   1:  PR[GP1:91,2] = PR[GP1:90,2] + 17.555;
   1:L PR[91] R[100]mm/sec CNT100;
   1:  PR[GP1:91,1] = PR[GP1:90,1] + 68.988;
   1:  PR[GP1:91,2] = PR[GP1:90,2] + 18.519;
   1:L PR[91] R[100]mm/sec CNT100;
   1:  PR[GP1:91,1] = PR[GP1:90,1] + 65.480;
   1:  PR[GP1:91,2] = PR[GP1:90,2] + 23.094;
   1:L PR[91] R[100]mm/sec CNT100;
   1:  PR[GP1:91,1] = PR[GP1:90,1] + 60.307;
   1:  PR[GP1:91,2] = PR[GP1:90,2] + 27.735;
   1:L PR[91] R[100]mm/sec CNT100;
   1:  PR[GP1:91,1] = PR[GP1:90,1] + 55.410;
   1:  PR[GP1:91,2] = PR[GP1:90,2] + 30.688;
   1:L PR[91] R[100]mm/sec CNT100;
   1:  PR[GP1:91,1] = PR[GP1:90,1] + 49.981;
   1:  PR[GP1:91,2] = PR[GP1:90,2] + 32.704;
   1:L PR[91] R[100]mm/sec CNT100;
   1:  PR[GP1:91,1] = PR[GP1:90,1] + 48.884;
   1:  PR[GP1:91,2] = PR[GP1:90,2] + 33.180;
   1:L PR[91] R[100]mm/sec CNT100;
   1:  PR[GP1:91,1] = PR[GP1:90,1] + 43.284;
   1:  PR[GP1:91,2] = PR[GP1:90,2] + 34.134;
   1:L PR[91] R[100]mm/sec CNT100;
   1:  PR[GP1:91,1] = PR[GP1:90,1] + 41.949;
   1:  PR[GP1:91,2] = PR[GP1:90,2] + 34.234;
   1:L PR[91] R[100]mm/sec CNT100;
   1:  PR[GP1:91,1] = PR[GP1:90,1] + 36.318;
   1:  PR[GP1:91,2] = PR[GP1:90,2] + 34.132;
   1:L PR[91] R[100]mm/sec CNT100;
   1:  PR[GP1:91,1] = PR[GP1:90,1] + 30.791;
   1:  PR[GP1:91,2] = PR[GP1:90,2] + 32.982;
   1:L PR[91] R[100]mm/sec CNT100;
   1:  PR[GP1:91,1] = PR[GP1:90,1] + 29.393;
   1:  PR[GP1:91,2] = PR[GP1:90,2] + 32.616;
   1:L PR[91] R[100]mm/sec CNT100;
   1:  PR[GP1:91,1] = PR[GP1:90,1] + 24.268;
   1:  PR[GP1:91,2] = PR[GP1:90,2] + 30.497;
   1:L PR[91] R[100]mm/sec CNT100;
   1:  PR[GP1:91,1] = PR[GP1:90,1] + 18.293;
   1:  PR[GP1:91,2] = PR[GP1:90,2] + 26.578;
   1:L PR[91] R[100]mm/sec CNT100;
   1:  PR[GP1:91,1] = PR[GP1:90,1] + 14.361;
   1:  PR[GP1:91,2] = PR[GP1:90,2] + 22.795;
   1:L PR[91] R[100]mm/sec CNT100;
   1:  PR[GP1:91,1] = PR[GP1:90,1] + 11.161;
   1:  PR[GP1:91,2] = PR[GP1:90,2] + 18.294;
   1:L PR[91] R[100]mm/sec CNT100;
   1:  PR[GP1:91,1] = PR[GP1:90,1] + 10.144;
   1:  PR[GP1:91,2] = PR[GP1:90,2] + 16.966;
   1:L PR[91] R[100]mm/sec CNT100;
   1:  PR[GP1:91,1] = PR[GP1:90,1] + 7.887;
   1:  PR[GP1:91,2] = PR[GP1:90,2] + 12.055;
   1:L PR[91] R[100]mm/sec CNT100;
   1:  PR[GP1:91,1] = PR[GP1:90,1] + 7.315;
   1:  PR[GP1:91,2] = PR[GP1:90,2] + 10.330;
   1:L PR[91] R[100]mm/sec CNT100;
   1:  PR[GP1:91,1] = PR[GP1:90,1] + 6.110;
   1:  PR[GP1:91,2] = PR[GP1:90,2] + 5.493;
   1:L PR[91] R[100]mm/sec CNT100;
   1:  PR[GP1:91,1] = PR[GP1:90,1] + 6.265;
   1:  PR[GP1:91,2] = PR[GP1:90,2] + 5.404;
   1:L PR[91] R[100]mm/sec CNT100;
   1:  PR[GP1:91,1] = PR[GP1:90,1] + 4.352;
   1:  PR[GP1:91,2] = PR[GP1:90,2] + 1.921;
   1:L PR[91] R[100]mm/sec CNT100;
   1:  PR[GP1:91,1] = PR[GP1:90,1] + 4.139;
   1:  PR[GP1:91,2] = PR[GP1:90,2] + 1.690;
   1:L PR[91] R[100]mm/sec CNT100;
   1:  PR[GP1:91,1] = PR[GP1:90,1] + 3.838;
   1:  PR[GP1:91,2] = PR[GP1:90,2] + 1.482;
   1:L PR[91] R[100]mm/sec CNT100;
   1:  PR[GP1:91,1] = PR[GP1:90,1] + 1.067;
   1:  PR[GP1:91,2] = PR[GP1:90,2] + 0.455;
   1:L PR[91] R[100]mm/sec CNT100;
   1:  PR[GP1:91,1] = PR[GP1:90,1] + 0.591;
   1:  PR[GP1:91,2] = PR[GP1:90,2] + 0.328;
   1:L PR[91] R[100]mm/sec CNT100;
   1:  PR[GP1:91,1] = PR[GP1:90,1] + -0.408;
   1:L PR[91] R[100]mm/sec CNT100;
   1:  ! -- Layer/Ebene 16 -- !;
   1:  PR[91] = PR[90];
   1:  PR[GP1:91,1] = PR[GP1:90,1] + -1.944;
   1:  PR[GP1:91,2] = PR[GP1:90,2] + 0.906;
   1:  PR[GP1:91,3] = PR[GP1:90,3] + 10.065;
   1:L PR[91] R[100]mm/sec CNT100;
   1:  PR[GP1:91,1] = PR[GP1:90,1] + -2.665;
   1:  PR[GP1:91,2] = PR[GP1:90,2] + 1.194;
   1:L PR[91] R[100]mm/sec CNT100;
   1:  PR[GP1:91,1] = PR[GP1:90,1] + -2.731;
   1:  PR[GP1:91,2] = PR[GP1:90,2] + 1.197;
   1:L PR[91] R[100]mm/sec CNT100;
   1:  PR[GP1:91,1] = PR[GP1:90,1] + -3.897;
   1:  PR[GP1:91,2] = PR[GP1:90,2] + 1.658;
   1:L PR[91] R[100]mm/sec CNT100;
   1:  PR[GP1:91,1] = PR[GP1:90,1] + -5.226;
   1:  PR[GP1:91,2] = PR[GP1:90,2] + 4.059;
   1:L PR[91] R[100]mm/sec CNT100;
   1:  PR[GP1:91,1] = PR[GP1:90,1] + -6.062;
   1:  PR[GP1:91,2] = PR[GP1:90,2] + 5.392;
   1:L PR[91] R[100]mm/sec CNT100;
   1:  PR[GP1:91,1] = PR[GP1:90,1] + -5.854;
   1:  PR[GP1:91,2] = PR[GP1:90,2] + 5.510;
   1:L PR[91] R[100]mm/sec CNT100;
   1:  PR[GP1:91,1] = PR[GP1:90,1] + -6.919;
   1:  PR[GP1:91,2] = PR[GP1:90,2] + 9.788;
   1:L PR[91] R[100]mm/sec CNT100;
   1:  PR[GP1:91,1] = PR[GP1:90,1] + -7.804;
   1:  PR[GP1:91,2] = PR[GP1:90,2] + 12.458;
   1:L PR[91] R[100]mm/sec CNT100;
   1:  PR[GP1:91,1] = PR[GP1:90,1] + -9.839;
   1:  PR[GP1:91,2] = PR[GP1:90,2] + 16.883;
   1:L PR[91] R[100]mm/sec CNT100;
   1:  PR[GP1:91,1] = PR[GP1:90,1] + -12.674;
   1:  PR[GP1:91,2] = PR[GP1:90,2] + 20.871;
   1:L PR[91] R[100]mm/sec CNT100;
   1:  PR[GP1:91,1] = PR[GP1:90,1] + -14.304;
   1:  PR[GP1:91,2] = PR[GP1:90,2] + 23.006;
   1:L PR[91] R[100]mm/sec CNT100;
   1:  PR[GP1:91,1] = PR[GP1:90,1] + -17.875;
   1:  PR[GP1:91,2] = PR[GP1:90,2] + 26.441;
   1:L PR[91] R[100]mm/sec CNT100;
   1:  PR[GP1:91,1] = PR[GP1:90,1] + -22.062;
   1:  PR[GP1:91,2] = PR[GP1:90,2] + 29.178;
   1:L PR[91] R[100]mm/sec CNT100;
   1:  PR[GP1:91,1] = PR[GP1:90,1] + -24.170;
   1:  PR[GP1:91,2] = PR[GP1:90,2] + 30.576;
   1:L PR[91] R[100]mm/sec CNT100;
   1:  PR[GP1:91,1] = PR[GP1:90,1] + -28.843;
   1:  PR[GP1:91,2] = PR[GP1:90,2] + 32.508;
   1:L PR[91] R[100]mm/sec CNT100;
   1:  PR[GP1:91,1] = PR[GP1:90,1] + -33.865;
   1:  PR[GP1:91,2] = PR[GP1:90,2] + 33.553;
   1:L PR[91] R[100]mm/sec CNT100;
   1:  PR[GP1:91,1] = PR[GP1:90,1] + -36.143;
   1:  PR[GP1:91,2] = PR[GP1:90,2] + 34.143;
   1:L PR[91] R[100]mm/sec CNT100;
   1:  PR[GP1:91,1] = PR[GP1:90,1] + -41.327;
   1:  PR[GP1:91,2] = PR[GP1:90,2] + 34.237;
   1:L PR[91] R[100]mm/sec CNT100;
   1:  PR[GP1:91,1] = PR[GP1:90,1] + -43.399;
   1:  PR[GP1:91,2] = PR[GP1:90,2] + 34.081;
   1:L PR[91] R[100]mm/sec CNT100;
   1:  PR[GP1:91,1] = PR[GP1:90,1] + -48.621;
   1:  PR[GP1:91,2] = PR[GP1:90,2] + 33.191;
   1:L PR[91] R[100]mm/sec CNT100;
   1:  PR[GP1:91,1] = PR[GP1:90,1] + -53.599;
   1:  PR[GP1:91,2] = PR[GP1:90,2] + 31.342;
   1:L PR[91] R[100]mm/sec CNT100;
   1:  PR[GP1:91,1] = PR[GP1:90,1] + -55.379;
   1:  PR[GP1:91,2] = PR[GP1:90,2] + 30.575;
   1:L PR[91] R[100]mm/sec CNT100;
   1:  PR[GP1:91,1] = PR[GP1:90,1] + -59.971;
   1:  PR[GP1:91,2] = PR[GP1:90,2] + 27.806;
   1:L PR[91] R[100]mm/sec CNT100;
   1:  PR[GP1:91,1] = PR[GP1:90,1] + -63.997;
   1:  PR[GP1:91,2] = PR[GP1:90,2] + 24.207;
   1:L PR[91] R[100]mm/sec CNT100;
   1:  PR[GP1:91,1] = PR[GP1:90,1] + -65.346;
   1:  PR[GP1:91,2] = PR[GP1:90,2] + 22.977;
   1:L PR[91] R[100]mm/sec CNT100;
   1:  PR[GP1:91,1] = PR[GP1:90,1] + -68.635;
   1:  PR[GP1:91,2] = PR[GP1:90,2] + 18.689;
   1:L PR[91] R[100]mm/sec CNT100;
   1:  PR[GP1:91,1] = PR[GP1:90,1] + -71.099;
   1:  PR[GP1:91,2] = PR[GP1:90,2] + 13.808;
   1:L PR[91] R[100]mm/sec CNT100;
   1:  PR[GP1:91,1] = PR[GP1:90,1] + -71.933;
   1:  PR[GP1:91,2] = PR[GP1:90,2] + 12.276;
   1:L PR[91] R[100]mm/sec CNT100;
   1:  PR[GP1:91,1] = PR[GP1:90,1] + -73.434;
   1:  PR[GP1:91,2] = PR[GP1:90,2] + 7.063;
   1:L PR[91] R[100]mm/sec CNT100;
   1:  PR[GP1:91,1] = PR[GP1:90,1] + -73.949;
   1:  PR[GP1:91,2] = PR[GP1:90,2] + 1.575;
   1:L PR[91] R[100]mm/sec CNT100;
   1:  PR[GP1:91,1] = PR[GP1:90,1] + -74.227;
   1:  PR[GP1:91,2] = PR[GP1:90,2] + -0.094;
   1:L PR[91] R[100]mm/sec CNT100;
   1:  PR[GP1:91,1] = PR[GP1:90,1] + -73.715;
   1:  PR[GP1:91,2] = PR[GP1:90,2] + -5.552;
   1:L PR[91] R[100]mm/sec CNT100;
   1:  PR[GP1:91,1] = PR[GP1:90,1] + -73.440;
   1:  PR[GP1:91,2] = PR[GP1:90,2] + -7.186;
   1:L PR[91] R[100]mm/sec CNT100;
   1:  PR[GP1:91,1] = PR[GP1:90,1] + -71.930;
   1:  PR[GP1:91,2] = PR[GP1:90,2] + -12.429;
   1:L PR[91] R[100]mm/sec CNT100;
   1:  PR[GP1:91,1] = PR[GP1:90,1] + -69.461;
   1:  PR[GP1:91,2] = PR[GP1:90,2] + -17.322;
   1:L PR[91] R[100]mm/sec CNT100;
   1:  PR[GP1:91,1] = PR[GP1:90,1] + -68.641;
   1:  PR[GP1:91,2] = PR[GP1:90,2] + -18.825;
   1:L PR[91] R[100]mm/sec CNT100;
   1:  PR[GP1:91,1] = PR[GP1:90,1] + -65.348;
   1:  PR[GP1:91,2] = PR[GP1:90,2] + -23.119;
   1:L PR[91] R[100]mm/sec CNT100;
   1:  PR[GP1:91,1] = PR[GP1:90,1] + -61.277;
   1:  PR[GP1:91,2] = PR[GP1:90,2] + -26.759;
   1:L PR[91] R[100]mm/sec CNT100;
   1:  PR[GP1:91,1] = PR[GP1:90,1] + -59.968;
   1:  PR[GP1:91,2] = PR[GP1:90,2] + -27.952;
   1:L PR[91] R[100]mm/sec CNT100;
   1:  PR[GP1:91,1] = PR[GP1:90,1] + -55.392;
   1:  PR[GP1:91,2] = PR[GP1:90,2] + -30.711;
   1:L PR[91] R[100]mm/sec CNT100;
   1:  PR[GP1:91,1] = PR[GP1:90,1] + -50.312;
   1:  PR[GP1:91,2] = PR[GP1:90,2] + -32.598;
   1:L PR[91] R[100]mm/sec CNT100;
   1:  PR[GP1:91,1] = PR[GP1:90,1] + -48.605;
   1:  PR[GP1:91,2] = PR[GP1:90,2] + -33.338;
   1:L PR[91] R[100]mm/sec CNT100;
   1:  PR[GP1:91,1] = PR[GP1:90,1] + -43.399;
   1:  PR[GP1:91,2] = PR[GP1:90,2] + -34.225;
   1:L PR[91] R[100]mm/sec CNT100;
   1:  PR[GP1:91,1] = PR[GP1:90,1] + -41.327;
   1:  PR[GP1:91,2] = PR[GP1:90,2] + -34.381;
   1:L PR[91] R[100]mm/sec CNT100;
   1:  PR[GP1:91,1] = PR[GP1:90,1] + -36.128;
   1:  PR[GP1:91,2] = PR[GP1:90,2] + -34.287;
   1:L PR[91] R[100]mm/sec CNT100;
   1:  PR[GP1:91,1] = PR[GP1:90,1] + -31.025;
   1:  PR[GP1:91,2] = PR[GP1:90,2] + -33.225;
   1:L PR[91] R[100]mm/sec CNT100;
   1:  PR[GP1:91,1] = PR[GP1:90,1] + -28.857;
   1:  PR[GP1:91,2] = PR[GP1:90,2] + -32.658;
   1:L PR[91] R[100]mm/sec CNT100;
   1:  PR[GP1:91,1] = PR[GP1:90,1] + -24.168;
   1:  PR[GP1:91,2] = PR[GP1:90,2] + -30.719;
   1:L PR[91] R[100]mm/sec CNT100;
   1:  PR[GP1:91,1] = PR[GP1:90,1] + -19.889;
   1:  PR[GP1:91,2] = PR[GP1:90,2] + -27.922;
   1:L PR[91] R[100]mm/sec CNT100;
   1:  PR[GP1:91,1] = PR[GP1:90,1] + -17.877;
   1:  PR[GP1:91,2] = PR[GP1:90,2] + -26.586;
   1:L PR[91] R[100]mm/sec CNT100;
   1:  PR[GP1:91,1] = PR[GP1:90,1] + -14.312;
   1:  PR[GP1:91,2] = PR[GP1:90,2] + -23.157;
   1:L PR[91] R[100]mm/sec CNT100;
   1:  PR[GP1:91,1] = PR[GP1:90,1] + -11.409;
   1:  PR[GP1:91,2] = PR[GP1:90,2] + -19.073;
   1:L PR[91] R[100]mm/sec CNT100;
   1:  PR[GP1:91,1] = PR[GP1:90,1] + -9.834;
   1:  PR[GP1:91,2] = PR[GP1:90,2] + -17.017;
   1:L PR[91] R[100]mm/sec CNT100;
   1:  PR[GP1:91,1] = PR[GP1:90,1] + -7.804;
   1:  PR[GP1:91,2] = PR[GP1:90,2] + -12.602;
   1:L PR[91] R[100]mm/sec CNT100;
   1:  PR[GP1:91,1] = PR[GP1:90,1] + -6.920;
   1:  PR[GP1:91,2] = PR[GP1:90,2] + -9.932;
   1:L PR[91] R[100]mm/sec CNT100;
   1:  PR[GP1:91,1] = PR[GP1:90,1] + -5.853;
   1:  PR[GP1:91,2] = PR[GP1:90,2] + -5.647;
   1:L PR[91] R[100]mm/sec CNT100;
   1:  PR[GP1:91,1] = PR[GP1:90,1] + -6.015;
   1:  PR[GP1:91,2] = PR[GP1:90,2] + -5.553;
   1:L PR[91] R[100]mm/sec CNT100;
   1:  PR[GP1:91,1] = PR[GP1:90,1] + -5.443;
   1:  PR[GP1:91,2] = PR[GP1:90,2] + -4.453;
   1:L PR[91] R[100]mm/sec CNT100;
   1:  PR[GP1:91,1] = PR[GP1:90,1] + -4.161;
   1:  PR[GP1:91,2] = PR[GP1:90,2] + -2.137;
   1:L PR[91] R[100]mm/sec CNT100;
   1:  PR[GP1:91,1] = PR[GP1:90,1] + -3.886;
   1:  PR[GP1:91,2] = PR[GP1:90,2] + -1.839;
   1:L PR[91] R[100]mm/sec CNT100;
   1:  PR[GP1:91,1] = PR[GP1:90,1] + -3.487;
   1:  PR[GP1:91,2] = PR[GP1:90,2] + -1.563;
   1:L PR[91] R[100]mm/sec CNT100;
   1:  PR[GP1:91,1] = PR[GP1:90,1] + -1.027;
   1:  PR[GP1:91,2] = PR[GP1:90,2] + -0.651;
   1:L PR[91] R[100]mm/sec CNT100;
   1:  PR[GP1:91,1] = PR[GP1:90,1] + -0.354;
   1:  PR[GP1:91,2] = PR[GP1:90,2] + -0.472;
   1:L PR[91] R[100]mm/sec CNT100;
   1:  PR[GP1:91,1] = PR[GP1:90,1] + 0.597;
   1:L PR[91] R[100]mm/sec CNT100;
   1:  PR[GP1:91,1] = PR[GP1:90,1] + 2.156;
   1:  PR[GP1:91,2] = PR[GP1:90,2] + -1.050;
   1:L PR[91] R[100]mm/sec CNT100;
   1:  PR[GP1:91,1] = PR[GP1:90,1] + 2.878;
   1:  PR[GP1:91,2] = PR[GP1:90,2] + -1.338;
   1:L PR[91] R[100]mm/sec CNT100;
   1:  PR[GP1:91,1] = PR[GP1:90,1] + 2.944;
   1:  PR[GP1:91,2] = PR[GP1:90,2] + -1.341;
   1:L PR[91] R[100]mm/sec CNT100;
   1:  PR[GP1:91,1] = PR[GP1:90,1] + 4.110;
   1:  PR[GP1:91,2] = PR[GP1:90,2] + -1.802;
   1:L PR[91] R[100]mm/sec CNT100;
   1:  PR[GP1:91,1] = PR[GP1:90,1] + 5.439;
   1:  PR[GP1:91,2] = PR[GP1:90,2] + -4.204;
   1:L PR[91] R[100]mm/sec CNT100;
   1:  PR[GP1:91,1] = PR[GP1:90,1] + 6.274;
   1:  PR[GP1:91,2] = PR[GP1:90,2] + -5.534;
   1:L PR[91] R[100]mm/sec CNT100;
   1:  PR[GP1:91,1] = PR[GP1:90,1] + 6.067;
   1:  PR[GP1:91,2] = PR[GP1:90,2] + -5.652;
   1:L PR[91] R[100]mm/sec CNT100;
   1:  PR[GP1:91,1] = PR[GP1:90,1] + 7.133;
   1:  PR[GP1:91,2] = PR[GP1:90,2] + -9.933;
   1:L PR[91] R[100]mm/sec CNT100;
   1:  PR[GP1:91,1] = PR[GP1:90,1] + 8.017;
   1:  PR[GP1:91,2] = PR[GP1:90,2] + -12.601;
   1:L PR[91] R[100]mm/sec CNT100;
   1:  PR[GP1:91,1] = PR[GP1:90,1] + 10.052;
   1:  PR[GP1:91,2] = PR[GP1:90,2] + -17.026;
   1:L PR[91] R[100]mm/sec CNT100;
   1:  PR[GP1:91,1] = PR[GP1:90,1] + 12.887;
   1:  PR[GP1:91,2] = PR[GP1:90,2] + -21.014;
   1:L PR[91] R[100]mm/sec CNT100;
   1:  PR[GP1:91,1] = PR[GP1:90,1] + 14.517;
   1:  PR[GP1:91,2] = PR[GP1:90,2] + -23.150;
   1:L PR[91] R[100]mm/sec CNT100;
   1:  PR[GP1:91,1] = PR[GP1:90,1] + 18.088;
   1:  PR[GP1:91,2] = PR[GP1:90,2] + -26.584;
   1:L PR[91] R[100]mm/sec CNT100;
   1:  PR[GP1:91,1] = PR[GP1:90,1] + 22.275;
   1:  PR[GP1:91,2] = PR[GP1:90,2] + -29.321;
   1:L PR[91] R[100]mm/sec CNT100;
   1:  PR[GP1:91,1] = PR[GP1:90,1] + 24.383;
   1:  PR[GP1:91,2] = PR[GP1:90,2] + -30.720;
   1:L PR[91] R[100]mm/sec CNT100;
   1:  PR[GP1:91,1] = PR[GP1:90,1] + 29.056;
   1:  PR[GP1:91,2] = PR[GP1:90,2] + -32.652;
   1:L PR[91] R[100]mm/sec CNT100;
   1:  PR[GP1:91,1] = PR[GP1:90,1] + 34.078;
   1:  PR[GP1:91,2] = PR[GP1:90,2] + -33.697;
   1:L PR[91] R[100]mm/sec CNT100;
   1:  PR[GP1:91,1] = PR[GP1:90,1] + 36.356;
   1:  PR[GP1:91,2] = PR[GP1:90,2] + -34.287;
   1:L PR[91] R[100]mm/sec CNT100;
   1:  PR[GP1:91,1] = PR[GP1:90,1] + 41.540;
   1:  PR[GP1:91,2] = PR[GP1:90,2] + -34.381;
   1:L PR[91] R[100]mm/sec CNT100;
   1:  PR[GP1:91,1] = PR[GP1:90,1] + 43.612;
   1:  PR[GP1:91,2] = PR[GP1:90,2] + -34.225;
   1:L PR[91] R[100]mm/sec CNT100;
   1:  PR[GP1:91,1] = PR[GP1:90,1] + 48.834;
   1:  PR[GP1:91,2] = PR[GP1:90,2] + -33.335;
   1:L PR[91] R[100]mm/sec CNT100;
   1:  PR[GP1:91,1] = PR[GP1:90,1] + 53.812;
   1:  PR[GP1:91,2] = PR[GP1:90,2] + -31.486;
   1:L PR[91] R[100]mm/sec CNT100;
   1:  PR[GP1:91,1] = PR[GP1:90,1] + 55.592;
   1:  PR[GP1:91,2] = PR[GP1:90,2] + -30.720;
   1:L PR[91] R[100]mm/sec CNT100;
   1:  PR[GP1:91,1] = PR[GP1:90,1] + 60.184;
   1:  PR[GP1:91,2] = PR[GP1:90,2] + -27.951;
   1:L PR[91] R[100]mm/sec CNT100;
   1:  PR[GP1:91,1] = PR[GP1:90,1] + 64.210;
   1:  PR[GP1:91,2] = PR[GP1:90,2] + -24.351;
   1:L PR[91] R[100]mm/sec CNT100;
   1:  PR[GP1:91,1] = PR[GP1:90,1] + 65.559;
   1:  PR[GP1:91,2] = PR[GP1:90,2] + -23.121;
   1:L PR[91] R[100]mm/sec CNT100;
   1:  PR[GP1:91,1] = PR[GP1:90,1] + 68.849;
   1:  PR[GP1:91,2] = PR[GP1:90,2] + -18.832;
   1:L PR[91] R[100]mm/sec CNT100;
   1:  PR[GP1:91,1] = PR[GP1:90,1] + 71.312;
   1:  PR[GP1:91,2] = PR[GP1:90,2] + -13.951;
   1:L PR[91] R[100]mm/sec CNT100;
   1:  PR[GP1:91,1] = PR[GP1:90,1] + 72.146;
   1:  PR[GP1:91,2] = PR[GP1:90,2] + -12.420;
   1:L PR[91] R[100]mm/sec CNT100;
   1:  PR[GP1:91,1] = PR[GP1:90,1] + 73.647;
   1:  PR[GP1:91,2] = PR[GP1:90,2] + -7.208;
   1:L PR[91] R[100]mm/sec CNT100;
   1:  PR[GP1:91,1] = PR[GP1:90,1] + 74.162;
   1:  PR[GP1:91,2] = PR[GP1:90,2] + -1.720;
   1:L PR[91] R[100]mm/sec CNT100;
   1:  PR[GP1:91,1] = PR[GP1:90,1] + 74.440;
   1:  PR[GP1:91,2] = PR[GP1:90,2] + -0.050;
   1:L PR[91] R[100]mm/sec CNT100;
   1:  PR[GP1:91,1] = PR[GP1:90,1] + 73.929;
   1:  PR[GP1:91,2] = PR[GP1:90,2] + 5.408;
   1:L PR[91] R[100]mm/sec CNT100;
   1:  PR[GP1:91,1] = PR[GP1:90,1] + 73.654;
   1:  PR[GP1:91,2] = PR[GP1:90,2] + 7.042;
   1:L PR[91] R[100]mm/sec CNT100;
   1:  PR[GP1:91,1] = PR[GP1:90,1] + 72.144;
   1:  PR[GP1:91,2] = PR[GP1:90,2] + 12.286;
   1:L PR[91] R[100]mm/sec CNT100;
   1:  PR[GP1:91,1] = PR[GP1:90,1] + 69.674;
   1:  PR[GP1:91,2] = PR[GP1:90,2] + 17.179;
   1:L PR[91] R[100]mm/sec CNT100;
   1:  PR[GP1:91,1] = PR[GP1:90,1] + 68.854;
   1:  PR[GP1:91,2] = PR[GP1:90,2] + 18.681;
   1:L PR[91] R[100]mm/sec CNT100;
   1:  PR[GP1:91,1] = PR[GP1:90,1] + 65.561;
   1:  PR[GP1:91,2] = PR[GP1:90,2] + 22.975;
   1:L PR[91] R[100]mm/sec CNT100;
   1:  PR[GP1:91,1] = PR[GP1:90,1] + 61.490;
   1:  PR[GP1:91,2] = PR[GP1:90,2] + 26.615;
   1:L PR[91] R[100]mm/sec CNT100;
   1:  PR[GP1:91,1] = PR[GP1:90,1] + 60.181;
   1:  PR[GP1:91,2] = PR[GP1:90,2] + 27.808;
   1:L PR[91] R[100]mm/sec CNT100;
   1:  PR[GP1:91,1] = PR[GP1:90,1] + 55.605;
   1:  PR[GP1:91,2] = PR[GP1:90,2] + 30.568;
   1:L PR[91] R[100]mm/sec CNT100;
   1:  PR[GP1:91,1] = PR[GP1:90,1] + 50.526;
   1:  PR[GP1:91,2] = PR[GP1:90,2] + 32.455;
   1:L PR[91] R[100]mm/sec CNT100;
   1:  PR[GP1:91,1] = PR[GP1:90,1] + 48.818;
   1:  PR[GP1:91,2] = PR[GP1:90,2] + 33.194;
   1:L PR[91] R[100]mm/sec CNT100;
   1:  PR[GP1:91,1] = PR[GP1:90,1] + 43.612;
   1:  PR[GP1:91,2] = PR[GP1:90,2] + 34.081;
   1:L PR[91] R[100]mm/sec CNT100;
   1:  PR[GP1:91,1] = PR[GP1:90,1] + 41.540;
   1:  PR[GP1:91,2] = PR[GP1:90,2] + 34.237;
   1:L PR[91] R[100]mm/sec CNT100;
   1:  PR[GP1:91,1] = PR[GP1:90,1] + 36.341;
   1:  PR[GP1:91,2] = PR[GP1:90,2] + 34.143;
   1:L PR[91] R[100]mm/sec CNT100;
   1:  PR[GP1:91,1] = PR[GP1:90,1] + 31.238;
   1:  PR[GP1:91,2] = PR[GP1:90,2] + 33.081;
   1:L PR[91] R[100]mm/sec CNT100;
   1:  PR[GP1:91,1] = PR[GP1:90,1] + 29.070;
   1:  PR[GP1:91,2] = PR[GP1:90,2] + 32.514;
   1:L PR[91] R[100]mm/sec CNT100;
   1:  PR[GP1:91,1] = PR[GP1:90,1] + 24.381;
   1:  PR[GP1:91,2] = PR[GP1:90,2] + 30.575;
   1:L PR[91] R[100]mm/sec CNT100;
   1:  PR[GP1:91,1] = PR[GP1:90,1] + 20.102;
   1:  PR[GP1:91,2] = PR[GP1:90,2] + 27.777;
   1:L PR[91] R[100]mm/sec CNT100;
   1:  PR[GP1:91,1] = PR[GP1:90,1] + 18.089;
   1:  PR[GP1:91,2] = PR[GP1:90,2] + 26.442;
   1:L PR[91] R[100]mm/sec CNT100;
   1:  PR[GP1:91,1] = PR[GP1:90,1] + 14.525;
   1:  PR[GP1:91,2] = PR[GP1:90,2] + 23.013;
   1:L PR[91] R[100]mm/sec CNT100;
   1:  PR[GP1:91,1] = PR[GP1:90,1] + 11.622;
   1:  PR[GP1:91,2] = PR[GP1:90,2] + 18.929;
   1:L PR[91] R[100]mm/sec CNT100;
   1:  PR[GP1:91,1] = PR[GP1:90,1] + 10.047;
   1:  PR[GP1:91,2] = PR[GP1:90,2] + 16.872;
   1:L PR[91] R[100]mm/sec CNT100;
   1:  PR[GP1:91,1] = PR[GP1:90,1] + 8.017;
   1:  PR[GP1:91,2] = PR[GP1:90,2] + 12.457;
   1:L PR[91] R[100]mm/sec CNT100;
   1:  PR[GP1:91,1] = PR[GP1:90,1] + 7.133;
   1:  PR[GP1:91,2] = PR[GP1:90,2] + 9.788;
   1:L PR[91] R[100]mm/sec CNT100;
   1:  PR[GP1:91,1] = PR[GP1:90,1] + 6.066;
   1:  PR[GP1:91,2] = PR[GP1:90,2] + 5.505;
   1:L PR[91] R[100]mm/sec CNT100;
   1:  PR[GP1:91,1] = PR[GP1:90,1] + 6.229;
   1:  PR[GP1:91,2] = PR[GP1:90,2] + 5.411;
   1:L PR[91] R[100]mm/sec CNT100;
   1:  PR[GP1:91,1] = PR[GP1:90,1] + 5.656;
   1:  PR[GP1:91,2] = PR[GP1:90,2] + 4.309;
   1:L PR[91] R[100]mm/sec CNT100;
   1:  PR[GP1:91,1] = PR[GP1:90,1] + 4.374;
   1:  PR[GP1:91,2] = PR[GP1:90,2] + 1.994;
   1:L PR[91] R[100]mm/sec CNT100;
   1:  PR[GP1:91,1] = PR[GP1:90,1] + 4.100;
   1:  PR[GP1:91,2] = PR[GP1:90,2] + 1.695;
   1:L PR[91] R[100]mm/sec CNT100;
   1:  PR[GP1:91,1] = PR[GP1:90,1] + 3.700;
   1:  PR[GP1:91,2] = PR[GP1:90,2] + 1.419;
   1:L PR[91] R[100]mm/sec CNT100;
   1:  PR[GP1:91,1] = PR[GP1:90,1] + 1.240;
   1:  PR[GP1:91,2] = PR[GP1:90,2] + 0.507;
   1:L PR[91] R[100]mm/sec CNT100;
   1:  PR[GP1:91,1] = PR[GP1:90,1] + 0.567;
   1:  PR[GP1:91,2] = PR[GP1:90,2] + 0.328;
   1:L PR[91] R[100]mm/sec CNT100;
   1:  PR[GP1:91,1] = PR[GP1:90,1] + -0.384;
   1:L PR[91] R[100]mm/sec CNT100;
   1:  ! -- Layer/Ebene 17 -- !;
   1:  PR[91] = PR[90];
   1:  PR[GP1:91,1] = PR[GP1:90,1] + -1.293;
   1:  PR[GP1:91,2] = PR[GP1:90,2] + 0.674;
   1:  PR[GP1:91,3] = PR[GP1:90,3] + 10.675;
   1:L PR[91] R[100]mm/sec CNT100;
   1:  PR[GP1:91,1] = PR[GP1:90,1] + -2.295;
   1:  PR[GP1:91,2] = PR[GP1:90,2] + 1.073;
   1:L PR[91] R[100]mm/sec CNT100;
   1:  PR[GP1:91,1] = PR[GP1:90,1] + -2.383;
   1:  PR[GP1:91,2] = PR[GP1:90,2] + 1.077;
   1:L PR[91] R[100]mm/sec CNT100;
   1:  PR[GP1:91,1] = PR[GP1:90,1] + -3.852;
   1:  PR[GP1:91,2] = PR[GP1:90,2] + 1.658;
   1:L PR[91] R[100]mm/sec CNT100;
   1:  PR[GP1:91,1] = PR[GP1:90,1] + -4.985;
   1:  PR[GP1:91,2] = PR[GP1:90,2] + 3.706;
   1:L PR[91] R[100]mm/sec CNT100;
   1:  PR[GP1:91,1] = PR[GP1:90,1] + -5.006;
   1:  PR[GP1:91,2] = PR[GP1:90,2] + 3.724;
   1:L PR[91] R[100]mm/sec CNT100;
   1:  PR[GP1:91,1] = PR[GP1:90,1] + -6.034;
   1:  PR[GP1:91,2] = PR[GP1:90,2] + 5.395;
   1:L PR[91] R[100]mm/sec CNT100;
   1:  PR[GP1:91,1] = PR[GP1:90,1] + -5.810;
   1:  PR[GP1:91,2] = PR[GP1:90,2] + 5.521;
   1:L PR[91] R[100]mm/sec CNT100;
   1:  PR[GP1:91,1] = PR[GP1:90,1] + -6.737;
   1:  PR[GP1:91,2] = PR[GP1:90,2] + 9.246;
   1:L PR[91] R[100]mm/sec CNT100;
   1:  PR[GP1:91,1] = PR[GP1:90,1] + -7.935;
   1:  PR[GP1:91,2] = PR[GP1:90,2] + 12.860;
   1:L PR[91] R[100]mm/sec CNT100;
   1:  PR[GP1:91,1] = PR[GP1:90,1] + -9.742;
   1:  PR[GP1:91,2] = PR[GP1:90,2] + 16.790;
   1:L PR[91] R[100]mm/sec CNT100;
   1:  PR[GP1:91,1] = PR[GP1:90,1] + -12.261;
   1:  PR[GP1:91,2] = PR[GP1:90,2] + 20.334;
   1:L PR[91] R[100]mm/sec CNT100;
   1:  PR[GP1:91,1] = PR[GP1:90,1] + -14.468;
   1:  PR[GP1:91,2] = PR[GP1:90,2] + 23.224;
   1:L PR[91] R[100]mm/sec CNT100;
   1:  PR[GP1:91,1] = PR[GP1:90,1] + -17.670;
   1:  PR[GP1:91,2] = PR[GP1:90,2] + 26.303;
   1:L PR[91] R[100]mm/sec CNT100;
   1:  PR[GP1:91,1] = PR[GP1:90,1] + -21.429;
   1:  PR[GP1:91,2] = PR[GP1:90,2] + 28.760;
   1:L PR[91] R[100]mm/sec CNT100;
   1:  PR[GP1:91,1] = PR[GP1:90,1] + -24.284;
   1:  PR[GP1:91,2] = PR[GP1:90,2] + 30.654;
   1:L PR[91] R[100]mm/sec CNT100;
   1:  PR[GP1:91,1] = PR[GP1:90,1] + -28.521;
   1:  PR[GP1:91,2] = PR[GP1:90,2] + 32.406;
   1:L PR[91] R[100]mm/sec CNT100;
   1:  PR[GP1:91,1] = PR[GP1:90,1] + -33.080;
   1:  PR[GP1:91,2] = PR[GP1:90,2] + 33.355;
   1:L PR[91] R[100]mm/sec CNT100;
   1:  PR[GP1:91,1] = PR[GP1:90,1] + -36.166;
   1:  PR[GP1:91,2] = PR[GP1:90,2] + 34.154;
   1:L PR[91] R[100]mm/sec CNT100;
   1:  PR[GP1:91,1] = PR[GP1:90,1] + -40.917;
   1:  PR[GP1:91,2] = PR[GP1:90,2] + 34.240;
   1:L PR[91] R[100]mm/sec CNT100;
   1:  PR[GP1:91,1] = PR[GP1:90,1] + -43.727;
   1:  PR[GP1:91,2] = PR[GP1:90,2] + 34.029;
   1:L PR[91] R[100]mm/sec CNT100;
   1:  PR[GP1:91,1] = PR[GP1:90,1] + -48.556;
   1:  PR[GP1:91,2] = PR[GP1:90,2] + 33.206;
   1:L PR[91] R[100]mm/sec CNT100;
   1:  PR[GP1:91,1] = PR[GP1:90,1] + -53.159;
   1:  PR[GP1:91,2] = PR[GP1:90,2] + 31.496;
   1:L PR[91] R[100]mm/sec CNT100;
   1:  PR[GP1:91,1] = PR[GP1:90,1] + -55.574;
   1:  PR[GP1:91,2] = PR[GP1:90,2] + 30.455;
   1:L PR[91] R[100]mm/sec CNT100;
   1:  PR[GP1:91,1] = PR[GP1:90,1] + -59.847;
   1:  PR[GP1:91,2] = PR[GP1:90,2] + 27.879;
   1:L PR[91] R[100]mm/sec CNT100;
   1:  PR[GP1:91,1] = PR[GP1:90,1] + -63.595;
   1:  PR[GP1:91,2] = PR[GP1:90,2] + 24.527;
   1:L PR[91] R[100]mm/sec CNT100;
   1:  PR[GP1:91,1] = PR[GP1:90,1] + -65.427;
   1:  PR[GP1:91,2] = PR[GP1:90,2] + 22.858;
   1:L PR[91] R[100]mm/sec CNT100;
   1:  PR[GP1:91,1] = PR[GP1:90,1] + -68.501;
   1:  PR[GP1:91,2] = PR[GP1:90,2] + 18.850;
   1:L PR[91] R[100]mm/sec CNT100;
   1:  PR[GP1:91,1] = PR[GP1:90,1] + -70.805;
   1:  PR[GP1:91,2] = PR[GP1:90,2] + 14.284;
   1:L PR[91] R[100]mm/sec CNT100;
   1:  PR[GP1:91,1] = PR[GP1:90,1] + -71.938;
   1:  PR[GP1:91,2] = PR[GP1:90,2] + 12.204;
   1:L PR[91] R[100]mm/sec CNT100;
   1:  PR[GP1:91,1] = PR[GP1:90,1] + -73.345;
   1:  PR[GP1:91,2] = PR[GP1:90,2] + 7.320;
   1:L PR[91] R[100]mm/sec CNT100;
   1:  PR[GP1:91,1] = PR[GP1:90,1] + -73.828;
   1:  PR[GP1:91,2] = PR[GP1:90,2] + 2.173;
   1:L PR[91] R[100]mm/sec CNT100;
   1:  PR[GP1:91,1] = PR[GP1:90,1] + -74.206;
   1:  PR[GP1:91,2] = PR[GP1:90,2] + -0.094;
   1:L PR[91] R[100]mm/sec CNT100;
   1:  PR[GP1:91,1] = PR[GP1:90,1] + -73.725;
   1:  PR[GP1:91,2] = PR[GP1:90,2] + -5.224;
   1:L PR[91] R[100]mm/sec CNT100;
   1:  PR[GP1:91,1] = PR[GP1:90,1] + -73.351;
   1:  PR[GP1:91,2] = PR[GP1:90,2] + -7.443;
   1:L PR[91] R[100]mm/sec CNT100;
   1:  PR[GP1:91,1] = PR[GP1:90,1] + -71.936;
   1:  PR[GP1:91,2] = PR[GP1:90,2] + -12.358;
   1:L PR[91] R[100]mm/sec CNT100;
   1:  PR[GP1:91,1] = PR[GP1:90,1] + -69.621;
   1:  PR[GP1:91,2] = PR[GP1:90,2] + -16.946;
   1:L PR[91] R[100]mm/sec CNT100;
   1:  PR[GP1:91,1] = PR[GP1:90,1] + -68.507;
   1:  PR[GP1:91,2] = PR[GP1:90,2] + -18.986;
   1:L PR[91] R[100]mm/sec CNT100;
   1:  PR[GP1:91,1] = PR[GP1:90,1] + -65.429;
   1:  PR[GP1:91,2] = PR[GP1:90,2] + -23.000;
   1:L PR[91] R[100]mm/sec CNT100;
   1:  PR[GP1:91,1] = PR[GP1:90,1] + -61.621;
   1:  PR[GP1:91,2] = PR[GP1:90,2] + -26.404;
   1:L PR[91] R[100]mm/sec CNT100;
   1:  PR[GP1:91,1] = PR[GP1:90,1] + -59.845;
   1:  PR[GP1:91,2] = PR[GP1:90,2] + -28.024;
   1:L PR[91] R[100]mm/sec CNT100;
   1:  PR[GP1:91,1] = PR[GP1:90,1] + -55.587;
   1:  PR[GP1:91,2] = PR[GP1:90,2] + -30.591;
   1:L PR[91] R[100]mm/sec CNT100;
   1:  PR[GP1:91,1] = PR[GP1:90,1] + -50.857;
   1:  PR[GP1:91,2] = PR[GP1:90,2] + -32.349;
   1:L PR[91] R[100]mm/sec CNT100;
   1:  PR[GP1:91,1] = PR[GP1:90,1] + -48.540;
   1:  PR[GP1:91,2] = PR[GP1:90,2] + -33.353;
   1:L PR[91] R[100]mm/sec CNT100;
   1:  PR[GP1:91,1] = PR[GP1:90,1] + -43.727;
   1:  PR[GP1:91,2] = PR[GP1:90,2] + -34.173;
   1:L PR[91] R[100]mm/sec CNT100;
   1:  PR[GP1:91,1] = PR[GP1:90,1] + -40.917;
   1:  PR[GP1:91,2] = PR[GP1:90,2] + -34.384;
   1:L PR[91] R[100]mm/sec CNT100;
   1:  PR[GP1:91,1] = PR[GP1:90,1] + -36.151;
   1:  PR[GP1:91,2] = PR[GP1:90,2] + -34.297;
   1:L PR[91] R[100]mm/sec CNT100;
   1:  PR[GP1:91,1] = PR[GP1:90,1] + -31.472;
   1:  PR[GP1:91,2] = PR[GP1:90,2] + -33.324;
   1:L PR[91] R[100]mm/sec CNT100;
   1:  PR[GP1:91,1] = PR[GP1:90,1] + -28.535;
   1:  PR[GP1:91,2] = PR[GP1:90,2] + -32.556;
   1:L PR[91] R[100]mm/sec CNT100;
   1:  PR[GP1:91,1] = PR[GP1:90,1] + -24.282;
   1:  PR[GP1:91,2] = PR[GP1:90,2] + -30.797;
   1:L PR[91] R[100]mm/sec CNT100;
   1:  PR[GP1:91,1] = PR[GP1:90,1] + -20.398;
   1:  PR[GP1:91,2] = PR[GP1:90,2] + -28.258;
   1:L PR[91] R[100]mm/sec CNT100;
   1:  PR[GP1:91,1] = PR[GP1:90,1] + -17.672;
   1:  PR[GP1:91,2] = PR[GP1:90,2] + -26.449;
   1:L PR[91] R[100]mm/sec CNT100;
   1:  PR[GP1:91,1] = PR[GP1:90,1] + -14.476;
   1:  PR[GP1:91,2] = PR[GP1:90,2] + -23.375;
   1:L PR[91] R[100]mm/sec CNT100;
   1:  PR[GP1:91,1] = PR[GP1:90,1] + -11.869;
   1:  PR[GP1:91,2] = PR[GP1:90,2] + -19.708;
   1:L PR[91] R[100]mm/sec CNT100;
   1:  PR[GP1:91,1] = PR[GP1:90,1] + -9.737;
   1:  PR[GP1:91,2] = PR[GP1:90,2] + -16.924;
   1:L PR[91] R[100]mm/sec CNT100;
   1:  PR[GP1:91,1] = PR[GP1:90,1] + -7.935;
   1:  PR[GP1:91,2] = PR[GP1:90,2] + -13.004;
   1:L PR[91] R[100]mm/sec CNT100;
   1:  PR[GP1:91,1] = PR[GP1:90,1] + -6.738;
   1:  PR[GP1:91,2] = PR[GP1:90,2] + -9.391;
   1:L PR[91] R[100]mm/sec CNT100;
   1:  PR[GP1:91,1] = PR[GP1:90,1] + -5.808;
   1:  PR[GP1:91,2] = PR[GP1:90,2] + -5.659;
   1:L PR[91] R[100]mm/sec CNT100;
   1:  PR[GP1:91,1] = PR[GP1:90,1] + -5.990;
   1:  PR[GP1:91,2] = PR[GP1:90,2] + -5.553;
   1:L PR[91] R[100]mm/sec CNT100;
   1:  PR[GP1:91,1] = PR[GP1:90,1] + -5.313;
   1:  PR[GP1:91,2] = PR[GP1:90,2] + -4.250;
   1:L PR[91] R[100]mm/sec CNT100;
   1:  PR[GP1:91,1] = PR[GP1:90,1] + -4.184;
   1:  PR[GP1:91,2] = PR[GP1:90,2] + -2.210;
   1:L PR[91] R[100]mm/sec CNT100;
   1:  PR[GP1:91,1] = PR[GP1:90,1] + -3.846;
   1:  PR[GP1:91,2] = PR[GP1:90,2] + -1.844;
   1:L PR[91] R[100]mm/sec CNT100;
   1:  PR[GP1:91,1] = PR[GP1:90,1] + -3.349;
   1:  PR[GP1:91,2] = PR[GP1:90,2] + -1.501;
   1:L PR[91] R[100]mm/sec CNT100;
   1:  PR[GP1:91,1] = PR[GP1:90,1] + -1.200;
   1:  PR[GP1:91,2] = PR[GP1:90,2] + -0.704;
   1:L PR[91] R[100]mm/sec CNT100;
   1:  PR[GP1:91,1] = PR[GP1:90,1] + -0.329;
   1:  PR[GP1:91,2] = PR[GP1:90,2] + -0.472;
   1:L PR[91] R[100]mm/sec CNT100;
   1:  PR[GP1:91,1] = PR[GP1:90,1] + 0.573;
   1:L PR[91] R[100]mm/sec CNT100;
   1:  PR[GP1:91,1] = PR[GP1:90,1] + 1.506;
   1:  PR[GP1:91,2] = PR[GP1:90,2] + -0.818;
   1:L PR[91] R[100]mm/sec CNT100;
   1:  PR[GP1:91,1] = PR[GP1:90,1] + 2.508;
   1:  PR[GP1:91,2] = PR[GP1:90,2] + -1.217;
   1:L PR[91] R[100]mm/sec CNT100;
   1:  PR[GP1:91,1] = PR[GP1:90,1] + 2.596;
   1:  PR[GP1:91,2] = PR[GP1:90,2] + -1.221;
   1:L PR[91] R[100]mm/sec CNT100;
   1:  PR[GP1:91,1] = PR[GP1:90,1] + 4.065;
   1:  PR[GP1:91,2] = PR[GP1:90,2] + -1.802;
   1:L PR[91] R[100]mm/sec CNT100;
   1:  PR[GP1:91,1] = PR[GP1:90,1] + 5.199;
   1:  PR[GP1:91,2] = PR[GP1:90,2] + -3.850;
   1:L PR[91] R[100]mm/sec CNT100;
   1:  PR[GP1:91,1] = PR[GP1:90,1] + 5.219;
   1:  PR[GP1:91,2] = PR[GP1:90,2] + -3.869;
   1:L PR[91] R[100]mm/sec CNT100;
   1:  PR[GP1:91,1] = PR[GP1:90,1] + 6.246;
   1:  PR[GP1:91,2] = PR[GP1:90,2] + -5.537;
   1:L PR[91] R[100]mm/sec CNT100;
   1:  PR[GP1:91,1] = PR[GP1:90,1] + 6.023;
   1:  PR[GP1:91,2] = PR[GP1:90,2] + -5.664;
   1:L PR[91] R[100]mm/sec CNT100;
   1:  PR[GP1:91,1] = PR[GP1:90,1] + 6.951;
   1:  PR[GP1:91,2] = PR[GP1:90,2] + -9.391;
   1:L PR[91] R[100]mm/sec CNT100;
   1:  PR[GP1:91,1] = PR[GP1:90,1] + 8.148;
   1:  PR[GP1:91,2] = PR[GP1:90,2] + -13.003;
   1:L PR[91] R[100]mm/sec CNT100;
   1:  PR[GP1:91,1] = PR[GP1:90,1] + 9.955;
   1:  PR[GP1:91,2] = PR[GP1:90,2] + -16.932;
   1:L PR[91] R[100]mm/sec CNT100;
   1:  PR[GP1:91,1] = PR[GP1:90,1] + 12.474;
   1:  PR[GP1:91,2] = PR[GP1:90,2] + -20.476;
   1:L PR[91] R[100]mm/sec CNT100;
   1:  PR[GP1:91,1] = PR[GP1:90,1] + 14.681;
   1:  PR[GP1:91,2] = PR[GP1:90,2] + -23.367;
   1:L PR[91] R[100]mm/sec CNT100;
   1:  PR[GP1:91,1] = PR[GP1:90,1] + 17.883;
   1:  PR[GP1:91,2] = PR[GP1:90,2] + -26.447;
   1:L PR[91] R[100]mm/sec CNT100;
   1:  PR[GP1:91,1] = PR[GP1:90,1] + 21.641;
   1:  PR[GP1:91,2] = PR[GP1:90,2] + -28.904;
   1:L PR[91] R[100]mm/sec CNT100;
   1:  PR[GP1:91,1] = PR[GP1:90,1] + 24.497;
   1:  PR[GP1:91,2] = PR[GP1:90,2] + -30.798;
   1:L PR[91] R[100]mm/sec CNT100;
   1:  PR[GP1:91,1] = PR[GP1:90,1] + 28.733;
   1:  PR[GP1:91,2] = PR[GP1:90,2] + -32.550;
   1:L PR[91] R[100]mm/sec CNT100;
   1:  PR[GP1:91,1] = PR[GP1:90,1] + 33.293;
   1:  PR[GP1:91,2] = PR[GP1:90,2] + -33.498;
   1:L PR[91] R[100]mm/sec CNT100;
   1:  PR[GP1:91,1] = PR[GP1:90,1] + 36.379;
   1:  PR[GP1:91,2] = PR[GP1:90,2] + -34.298;
   1:L PR[91] R[100]mm/sec CNT100;
   1:  PR[GP1:91,1] = PR[GP1:90,1] + 41.130;
   1:  PR[GP1:91,2] = PR[GP1:90,2] + -34.384;
   1:L PR[91] R[100]mm/sec CNT100;
   1:  PR[GP1:91,1] = PR[GP1:90,1] + 43.940;
   1:  PR[GP1:91,2] = PR[GP1:90,2] + -34.173;
   1:L PR[91] R[100]mm/sec CNT100;
   1:  PR[GP1:91,1] = PR[GP1:90,1] + 48.769;
   1:  PR[GP1:91,2] = PR[GP1:90,2] + -33.350;
   1:L PR[91] R[100]mm/sec CNT100;
   1:  PR[GP1:91,1] = PR[GP1:90,1] + 53.372;
   1:  PR[GP1:91,2] = PR[GP1:90,2] + -31.640;
   1:L PR[91] R[100]mm/sec CNT100;
   1:  PR[GP1:91,1] = PR[GP1:90,1] + 55.787;
   1:  PR[GP1:91,2] = PR[GP1:90,2] + -30.600;
   1:L PR[91] R[100]mm/sec CNT100;
   1:  PR[GP1:91,1] = PR[GP1:90,1] + 60.060;
   1:  PR[GP1:91,2] = PR[GP1:90,2] + -28.023;
   1:L PR[91] R[100]mm/sec CNT100;
   1:  PR[GP1:91,1] = PR[GP1:90,1] + 63.809;
   1:  PR[GP1:91,2] = PR[GP1:90,2] + -24.671;
   1:L PR[91] R[100]mm/sec CNT100;
   1:  PR[GP1:91,1] = PR[GP1:90,1] + 65.640;
   1:  PR[GP1:91,2] = PR[GP1:90,2] + -23.002;
   1:L PR[91] R[100]mm/sec CNT100;
   1:  PR[GP1:91,1] = PR[GP1:90,1] + 68.715;
   1:  PR[GP1:91,2] = PR[GP1:90,2] + -18.994;
   1:L PR[91] R[100]mm/sec CNT100;
   1:  PR[GP1:91,1] = PR[GP1:90,1] + 71.019;
   1:  PR[GP1:91,2] = PR[GP1:90,2] + -14.428;
   1:L PR[91] R[100]mm/sec CNT100;
   1:  PR[GP1:91,1] = PR[GP1:90,1] + 72.152;
   1:  PR[GP1:91,2] = PR[GP1:90,2] + -12.349;
   1:L PR[91] R[100]mm/sec CNT100;
   1:  PR[GP1:91,1] = PR[GP1:90,1] + 73.558;
   1:  PR[GP1:91,2] = PR[GP1:90,2] + -7.465;
   1:L PR[91] R[100]mm/sec CNT100;
   1:  PR[GP1:91,1] = PR[GP1:90,1] + 74.041;
   1:  PR[GP1:91,2] = PR[GP1:90,2] + -2.317;
   1:L PR[91] R[100]mm/sec CNT100;
   1:  PR[GP1:91,1] = PR[GP1:90,1] + 74.419;
   1:  PR[GP1:91,2] = PR[GP1:90,2] + -0.050;
   1:L PR[91] R[100]mm/sec CNT100;
   1:  PR[GP1:91,1] = PR[GP1:90,1] + 73.938;
   1:  PR[GP1:91,2] = PR[GP1:90,2] + 5.080;
   1:L PR[91] R[100]mm/sec CNT100;
   1:  PR[GP1:91,1] = PR[GP1:90,1] + 73.564;
   1:  PR[GP1:91,2] = PR[GP1:90,2] + 7.300;
   1:L PR[91] R[100]mm/sec CNT100;
   1:  PR[GP1:91,1] = PR[GP1:90,1] + 72.149;
   1:  PR[GP1:91,2] = PR[GP1:90,2] + 12.215;
   1:L PR[91] R[100]mm/sec CNT100;
   1:  PR[GP1:91,1] = PR[GP1:90,1] + 69.834;
   1:  PR[GP1:91,2] = PR[GP1:90,2] + 16.802;
   1:L PR[91] R[100]mm/sec CNT100;
   1:  PR[GP1:91,1] = PR[GP1:90,1] + 68.721;
   1:  PR[GP1:91,2] = PR[GP1:90,2] + 18.842;
   1:L PR[91] R[100]mm/sec CNT100;
   1:  PR[GP1:91,1] = PR[GP1:90,1] + 65.642;
   1:  PR[GP1:91,2] = PR[GP1:90,2] + 22.856;
   1:L PR[91] R[100]mm/sec CNT100;
   1:  PR[GP1:91,1] = PR[GP1:90,1] + 61.834;
   1:  PR[GP1:91,2] = PR[GP1:90,2] + 26.260;
   1:L PR[91] R[100]mm/sec CNT100;
   1:  PR[GP1:91,1] = PR[GP1:90,1] + 60.058;
   1:  PR[GP1:91,2] = PR[GP1:90,2] + 27.881;
   1:L PR[91] R[100]mm/sec CNT100;
   1:  PR[GP1:91,1] = PR[GP1:90,1] + 55.800;
   1:  PR[GP1:91,2] = PR[GP1:90,2] + 30.448;
   1:L PR[91] R[100]mm/sec CNT100;
   1:  PR[GP1:91,1] = PR[GP1:90,1] + 51.070;
   1:  PR[GP1:91,2] = PR[GP1:90,2] + 32.205;
   1:L PR[91] R[100]mm/sec CNT100;
   1:  PR[GP1:91,1] = PR[GP1:90,1] + 48.753;
   1:  PR[GP1:91,2] = PR[GP1:90,2] + 33.209;
   1:L PR[91] R[100]mm/sec CNT100;
   1:  PR[GP1:91,1] = PR[GP1:90,1] + 43.940;
   1:  PR[GP1:91,2] = PR[GP1:90,2] + 34.029;
   1:L PR[91] R[100]mm/sec CNT100;
   1:  PR[GP1:91,1] = PR[GP1:90,1] + 41.130;
   1:  PR[GP1:91,2] = PR[GP1:90,2] + 34.240;
   1:L PR[91] R[100]mm/sec CNT100;
   1:  PR[GP1:91,1] = PR[GP1:90,1] + 36.364;
   1:  PR[GP1:91,2] = PR[GP1:90,2] + 34.153;
   1:L PR[91] R[100]mm/sec CNT100;
   1:  PR[GP1:91,1] = PR[GP1:90,1] + 31.685;
   1:  PR[GP1:91,2] = PR[GP1:90,2] + 33.180;
   1:L PR[91] R[100]mm/sec CNT100;
   1:  PR[GP1:91,1] = PR[GP1:90,1] + 28.747;
   1:  PR[GP1:91,2] = PR[GP1:90,2] + 32.411;
   1:L PR[91] R[100]mm/sec CNT100;
   1:  PR[GP1:91,1] = PR[GP1:90,1] + 24.495;
   1:  PR[GP1:91,2] = PR[GP1:90,2] + 30.653;
   1:L PR[91] R[100]mm/sec CNT100;
   1:  PR[GP1:91,1] = PR[GP1:90,1] + 20.610;
   1:  PR[GP1:91,2] = PR[GP1:90,2] + 28.114;
   1:L PR[91] R[100]mm/sec CNT100;
   1:  PR[GP1:91,1] = PR[GP1:90,1] + 17.884;
   1:  PR[GP1:91,2] = PR[GP1:90,2] + 26.304;
   1:L PR[91] R[100]mm/sec CNT100;
   1:  PR[GP1:91,1] = PR[GP1:90,1] + 14.688;
   1:  PR[GP1:91,2] = PR[GP1:90,2] + 23.230;
   1:L PR[91] R[100]mm/sec CNT100;
   1:  PR[GP1:91,1] = PR[GP1:90,1] + 12.082;
   1:  PR[GP1:91,2] = PR[GP1:90,2] + 19.563;
   1:L PR[91] R[100]mm/sec CNT100;
   1:  PR[GP1:91,1] = PR[GP1:90,1] + 9.950;
   1:  PR[GP1:91,2] = PR[GP1:90,2] + 16.779;
   1:L PR[91] R[100]mm/sec CNT100;
   1:  PR[GP1:91,1] = PR[GP1:90,1] + 8.148;
   1:  PR[GP1:91,2] = PR[GP1:90,2] + 12.859;
   1:L PR[91] R[100]mm/sec CNT100;
   1:  PR[GP1:91,1] = PR[GP1:90,1] + 6.951;
   1:  PR[GP1:91,2] = PR[GP1:90,2] + 9.246;
   1:L PR[91] R[100]mm/sec CNT100;
   1:  PR[GP1:91,1] = PR[GP1:90,1] + 6.022;
   1:  PR[GP1:91,2] = PR[GP1:90,2] + 5.517;
   1:L PR[91] R[100]mm/sec CNT100;
   1:  PR[GP1:91,1] = PR[GP1:90,1] + 6.204;
   1:  PR[GP1:91,2] = PR[GP1:90,2] + 5.411;
   1:L PR[91] R[100]mm/sec CNT100;
   1:  PR[GP1:91,1] = PR[GP1:90,1] + 5.526;
   1:  PR[GP1:91,2] = PR[GP1:90,2] + 4.106;
   1:L PR[91] R[100]mm/sec CNT100;
   1:  PR[GP1:91,1] = PR[GP1:90,1] + 4.397;
   1:  PR[GP1:91,2] = PR[GP1:90,2] + 2.066;
   1:L PR[91] R[100]mm/sec CNT100;
   1:  PR[GP1:91,1] = PR[GP1:90,1] + 4.060;
   1:  PR[GP1:91,2] = PR[GP1:90,2] + 1.700;
   1:L PR[91] R[100]mm/sec CNT100;
   1:  PR[GP1:91,1] = PR[GP1:90,1] + 3.562;
   1:  PR[GP1:91,2] = PR[GP1:90,2] + 1.357;
   1:L PR[91] R[100]mm/sec CNT100;
   1:  PR[GP1:91,1] = PR[GP1:90,1] + 1.413;
   1:  PR[GP1:91,2] = PR[GP1:90,2] + 0.560;
   1:L PR[91] R[100]mm/sec CNT100;
   1:  PR[GP1:91,1] = PR[GP1:90,1] + 0.542;
   1:  PR[GP1:91,2] = PR[GP1:90,2] + 0.328;
   1:L PR[91] R[100]mm/sec CNT100;
   1:  PR[GP1:91,1] = PR[GP1:90,1] + -0.360;
   1:L PR[91] R[100]mm/sec CNT100;
   1:  ! -- Layer/Ebene 18 -- !;
   1:  PR[91] = PR[90];
   1:  PR[GP1:91,1] = PR[GP1:90,1] + -1.924;
   1:  PR[GP1:91,2] = PR[GP1:90,2] + 0.953;
   1:  PR[GP1:91,3] = PR[GP1:90,3] + 11.285;
   1:L PR[91] R[100]mm/sec CNT100;
   1:  PR[GP1:91,1] = PR[GP1:90,1] + -2.036;
   1:  PR[GP1:91,2] = PR[GP1:90,2] + 0.958;
   1:L PR[91] R[100]mm/sec CNT100;
   1:  PR[GP1:91,1] = PR[GP1:90,1] + -3.807;
   1:  PR[GP1:91,2] = PR[GP1:90,2] + 1.658;
   1:L PR[91] R[100]mm/sec CNT100;
   1:  PR[GP1:91,1] = PR[GP1:90,1] + -4.784;
   1:  PR[GP1:91,2] = PR[GP1:90,2] + 3.424;
   1:L PR[91] R[100]mm/sec CNT100;
   1:  PR[GP1:91,1] = PR[GP1:90,1] + -4.813;
   1:  PR[GP1:91,2] = PR[GP1:90,2] + 3.450;
   1:L PR[91] R[100]mm/sec CNT100;
   1:  PR[GP1:91,1] = PR[GP1:90,1] + -6.010;
   1:  PR[GP1:91,2] = PR[GP1:90,2] + 5.395;
   1:L PR[91] R[100]mm/sec CNT100;
   1:  PR[GP1:91,1] = PR[GP1:90,1] + -5.766;
   1:  PR[GP1:91,2] = PR[GP1:90,2] + 5.533;
   1:L PR[91] R[100]mm/sec CNT100;
   1:  PR[GP1:91,1] = PR[GP1:90,1] + -6.555;
   1:  PR[GP1:91,2] = PR[GP1:90,2] + 8.705;
   1:L PR[91] R[100]mm/sec CNT100;
   1:  PR[GP1:91,1] = PR[GP1:90,1] + -8.066;
   1:  PR[GP1:91,2] = PR[GP1:90,2] + 13.262;
   1:L PR[91] R[100]mm/sec CNT100;
   1:  PR[GP1:91,1] = PR[GP1:90,1] + -9.645;
   1:  PR[GP1:91,2] = PR[GP1:90,2] + 16.697;
   1:L PR[91] R[100]mm/sec CNT100;
   1:  PR[GP1:91,1] = PR[GP1:90,1] + -11.848;
   1:  PR[GP1:91,2] = PR[GP1:90,2] + 19.796;
   1:L PR[91] R[100]mm/sec CNT100;
   1:  PR[GP1:91,1] = PR[GP1:90,1] + -14.632;
   1:  PR[GP1:91,2] = PR[GP1:90,2] + 23.441;
   1:L PR[91] R[100]mm/sec CNT100;
   1:  PR[GP1:91,1] = PR[GP1:90,1] + -17.465;
   1:  PR[GP1:91,2] = PR[GP1:90,2] + 26.166;
   1:L PR[91] R[100]mm/sec CNT100;
   1:  PR[GP1:91,1] = PR[GP1:90,1] + -20.795;
   1:  PR[GP1:91,2] = PR[GP1:90,2] + 28.343;
   1:L PR[91] R[100]mm/sec CNT100;
   1:  PR[GP1:91,1] = PR[GP1:90,1] + -24.397;
   1:  PR[GP1:91,2] = PR[GP1:90,2] + 30.732;
   1:L PR[91] R[100]mm/sec CNT100;
   1:  PR[GP1:91,1] = PR[GP1:90,1] + -28.198;
   1:  PR[GP1:91,2] = PR[GP1:90,2] + 32.304;
   1:L PR[91] R[100]mm/sec CNT100;
   1:  PR[GP1:91,1] = PR[GP1:90,1] + -32.295;
   1:  PR[GP1:91,2] = PR[GP1:90,2] + 33.156;
   1:L PR[91] R[100]mm/sec CNT100;
   1:  PR[GP1:91,1] = PR[GP1:90,1] + -36.189;
   1:  PR[GP1:91,2] = PR[GP1:90,2] + 34.165;
   1:L PR[91] R[100]mm/sec CNT100;
   1:  PR[GP1:91,1] = PR[GP1:90,1] + -40.507;
   1:  PR[GP1:91,2] = PR[GP1:90,2] + 34.243;
   1:L PR[91] R[100]mm/sec CNT100;
   1:  PR[GP1:91,1] = PR[GP1:90,1] + -44.055;
   1:  PR[GP1:91,2] = PR[GP1:90,2] + 33.976;
   1:L PR[91] R[100]mm/sec CNT100;
   1:  PR[GP1:91,1] = PR[GP1:90,1] + -48.490;
   1:  PR[GP1:91,2] = PR[GP1:90,2] + 33.220;
   1:L PR[91] R[100]mm/sec CNT100;
   1:  PR[GP1:91,1] = PR[GP1:90,1] + -52.720;
   1:  PR[GP1:91,2] = PR[GP1:90,2] + 31.649;
   1:L PR[91] R[100]mm/sec CNT100;
   1:  PR[GP1:91,1] = PR[GP1:90,1] + -55.769;
   1:  PR[GP1:91,2] = PR[GP1:90,2] + 30.335;
   1:L PR[91] R[100]mm/sec CNT100;
   1:  PR[GP1:91,1] = PR[GP1:90,1] + -59.724;
   1:  PR[GP1:91,2] = PR[GP1:90,2] + 27.951;
   1:L PR[91] R[100]mm/sec CNT100;
   1:  PR[GP1:91,1] = PR[GP1:90,1] + -63.194;
   1:  PR[GP1:91,2] = PR[GP1:90,2] + 24.848;
   1:L PR[91] R[100]mm/sec CNT100;
   1:  PR[GP1:91,1] = PR[GP1:90,1] + -65.508;
   1:  PR[GP1:91,2] = PR[GP1:90,2] + 22.739;
   1:L PR[91] R[100]mm/sec CNT100;
   1:  PR[GP1:91,1] = PR[GP1:90,1] + -68.368;
   1:  PR[GP1:91,2] = PR[GP1:90,2] + 19.011;
   1:L PR[91] R[100]mm/sec CNT100;
   1:  PR[GP1:91,1] = PR[GP1:90,1] + -70.512;
   1:  PR[GP1:91,2] = PR[GP1:90,2] + 14.761;
   1:L PR[91] R[100]mm/sec CNT100;
   1:  PR[GP1:91,1] = PR[GP1:90,1] + -71.944;
   1:  PR[GP1:91,2] = PR[GP1:90,2] + 12.133;
   1:L PR[91] R[100]mm/sec CNT100;
   1:  PR[GP1:91,1] = PR[GP1:90,1] + -73.256;
   1:  PR[GP1:91,2] = PR[GP1:90,2] + 7.577;
   1:L PR[91] R[100]mm/sec CNT100;
   1:  PR[GP1:91,1] = PR[GP1:90,1] + -73.707;
   1:  PR[GP1:91,2] = PR[GP1:90,2] + 2.770;
   1:L PR[91] R[100]mm/sec CNT100;
   1:  PR[GP1:91,1] = PR[GP1:90,1] + -74.184;
   1:  PR[GP1:91,2] = PR[GP1:90,2] + -0.094;
   1:L PR[91] R[100]mm/sec CNT100;
   1:  PR[GP1:91,1] = PR[GP1:90,1] + -73.734;
   1:  PR[GP1:91,2] = PR[GP1:90,2] + -4.895;
   1:L PR[91] R[100]mm/sec CNT100;
   1:  PR[GP1:91,1] = PR[GP1:90,1] + -73.262;
   1:  PR[GP1:91,2] = PR[GP1:90,2] + -7.700;
   1:L PR[91] R[100]mm/sec CNT100;
   1:  PR[GP1:91,1] = PR[GP1:90,1] + -71.941;
   1:  PR[GP1:91,2] = PR[GP1:90,2] + -12.286;
   1:L PR[91] R[100]mm/sec CNT100;
   1:  PR[GP1:91,1] = PR[GP1:90,1] + -69.780;
   1:  PR[GP1:91,2] = PR[GP1:90,2] + -16.569;
   1:L PR[91] R[100]mm/sec CNT100;
   1:  PR[GP1:91,1] = PR[GP1:90,1] + -68.373;
   1:  PR[GP1:91,2] = PR[GP1:90,2] + -19.148;
   1:L PR[91] R[100]mm/sec CNT100;
   1:  PR[GP1:91,1] = PR[GP1:90,1] + -65.510;
   1:  PR[GP1:91,2] = PR[GP1:90,2] + -22.881;
   1:L PR[91] R[100]mm/sec CNT100;
   1:  PR[GP1:91,1] = PR[GP1:90,1] + -61.966;
   1:  PR[GP1:91,2] = PR[GP1:90,2] + -26.050;
   1:L PR[91] R[100]mm/sec CNT100;
   1:  PR[GP1:91,1] = PR[GP1:90,1] + -59.721;
   1:  PR[GP1:91,2] = PR[GP1:90,2] + -28.096;
   1:L PR[91] R[100]mm/sec CNT100;
   1:  PR[GP1:91,1] = PR[GP1:90,1] + -55.783;
   1:  PR[GP1:91,2] = PR[GP1:90,2] + -30.471;
   1:L PR[91] R[100]mm/sec CNT100;
   1:  PR[GP1:91,1] = PR[GP1:90,1] + -51.401;
   1:  PR[GP1:91,2] = PR[GP1:90,2] + -32.099;
   1:L PR[91] R[100]mm/sec CNT100;
   1:  PR[GP1:91,1] = PR[GP1:90,1] + -48.474;
   1:  PR[GP1:91,2] = PR[GP1:90,2] + -33.367;
   1:L PR[91] R[100]mm/sec CNT100;
   1:  PR[GP1:91,1] = PR[GP1:90,1] + -44.055;
   1:  PR[GP1:91,2] = PR[GP1:90,2] + -34.120;
   1:L PR[91] R[100]mm/sec CNT100;
   1:  PR[GP1:91,1] = PR[GP1:90,1] + -40.507;
   1:  PR[GP1:91,2] = PR[GP1:90,2] + -34.387;
   1:L PR[91] R[100]mm/sec CNT100;
   1:  PR[GP1:91,1] = PR[GP1:90,1] + -36.175;
   1:  PR[GP1:91,2] = PR[GP1:90,2] + -34.308;
   1:L PR[91] R[100]mm/sec CNT100;
   1:  PR[GP1:91,1] = PR[GP1:90,1] + -31.919;
   1:  PR[GP1:91,2] = PR[GP1:90,2] + -33.423;
   1:L PR[91] R[100]mm/sec CNT100;
   1:  PR[GP1:91,1] = PR[GP1:90,1] + -28.212;
   1:  PR[GP1:91,2] = PR[GP1:90,2] + -32.454;
   1:L PR[91] R[100]mm/sec CNT100;
   1:  PR[GP1:91,1] = PR[GP1:90,1] + -24.396;
   1:  PR[GP1:91,2] = PR[GP1:90,2] + -30.876;
   1:L PR[91] R[100]mm/sec CNT100;
   1:  PR[GP1:91,1] = PR[GP1:90,1] + -20.907;
   1:  PR[GP1:91,2] = PR[GP1:90,2] + -28.595;
   1:L PR[91] R[100]mm/sec CNT100;
   1:  PR[GP1:91,1] = PR[GP1:90,1] + -17.467;
   1:  PR[GP1:91,2] = PR[GP1:90,2] + -26.311;
   1:L PR[91] R[100]mm/sec CNT100;
   1:  PR[GP1:91,1] = PR[GP1:90,1] + -14.640;
   1:  PR[GP1:91,2] = PR[GP1:90,2] + -23.592;
   1:L PR[91] R[100]mm/sec CNT100;
   1:  PR[GP1:91,1] = PR[GP1:90,1] + -12.330;
   1:  PR[GP1:91,2] = PR[GP1:90,2] + -20.342;
   1:L PR[91] R[100]mm/sec CNT100;
   1:  PR[GP1:91,1] = PR[GP1:90,1] + -9.640;
   1:  PR[GP1:91,2] = PR[GP1:90,2] + -16.831;
   1:L PR[91] R[100]mm/sec CNT100;
   1:  PR[GP1:91,1] = PR[GP1:90,1] + -8.066;
   1:  PR[GP1:91,2] = PR[GP1:90,2] + -13.406;
   1:L PR[91] R[100]mm/sec CNT100;
   1:  PR[GP1:91,1] = PR[GP1:90,1] + -6.556;
   1:  PR[GP1:91,2] = PR[GP1:90,2] + -8.850;
   1:L PR[91] R[100]mm/sec CNT100;
   1:  PR[GP1:91,1] = PR[GP1:90,1] + -5.764;
   1:  PR[GP1:91,2] = PR[GP1:90,2] + -5.671;
   1:L PR[91] R[100]mm/sec CNT100;
   1:  PR[GP1:91,1] = PR[GP1:90,1] + -5.966;
   1:  PR[GP1:91,2] = PR[GP1:90,2] + -5.553;
   1:L PR[91] R[100]mm/sec CNT100;
   1:  PR[GP1:91,1] = PR[GP1:90,1] + -5.183;
   1:  PR[GP1:91,2] = PR[GP1:90,2] + -4.047;
   1:L PR[91] R[100]mm/sec CNT100;
   1:  PR[GP1:91,1] = PR[GP1:90,1] + -4.207;
   1:  PR[GP1:91,2] = PR[GP1:90,2] + -2.283;
   1:L PR[91] R[100]mm/sec CNT100;
   1:  PR[GP1:91,1] = PR[GP1:90,1] + -3.807;
   1:  PR[GP1:91,2] = PR[GP1:90,2] + -1.849;
   1:L PR[91] R[100]mm/sec CNT100;
   1:  PR[GP1:91,1] = PR[GP1:90,1] + -3.211;
   1:  PR[GP1:91,2] = PR[GP1:90,2] + -1.438;
   1:L PR[91] R[100]mm/sec CNT100;
   1:  PR[GP1:91,1] = PR[GP1:90,1] + -1.373;
   1:  PR[GP1:91,2] = PR[GP1:90,2] + -0.757;
   1:L PR[91] R[100]mm/sec CNT100;
   1:  PR[GP1:91,1] = PR[GP1:90,1] + -0.305;
   1:  PR[GP1:91,2] = PR[GP1:90,2] + -0.472;
   1:L PR[91] R[100]mm/sec CNT100;
   1:  PR[GP1:91,1] = PR[GP1:90,1] + 0.556;
   1:L PR[91] R[100]mm/sec CNT100;
   1:  PR[GP1:91,1] = PR[GP1:90,1] + 2.137;
   1:  PR[GP1:91,2] = PR[GP1:90,2] + -1.097;
   1:L PR[91] R[100]mm/sec CNT100;
   1:  PR[GP1:91,1] = PR[GP1:90,1] + 2.249;
   1:  PR[GP1:91,2] = PR[GP1:90,2] + -1.102;
   1:L PR[91] R[100]mm/sec CNT100;
   1:  PR[GP1:91,1] = PR[GP1:90,1] + 4.020;
   1:  PR[GP1:91,2] = PR[GP1:90,2] + -1.803;
   1:L PR[91] R[100]mm/sec CNT100;
   1:  PR[GP1:91,1] = PR[GP1:90,1] + 4.998;
   1:  PR[GP1:91,2] = PR[GP1:90,2] + -3.568;
   1:L PR[91] R[100]mm/sec CNT100;
   1:  PR[GP1:91,1] = PR[GP1:90,1] + 5.026;
   1:  PR[GP1:91,2] = PR[GP1:90,2] + -3.594;
   1:L PR[91] R[100]mm/sec CNT100;
   1:  PR[GP1:91,1] = PR[GP1:90,1] + 6.222;
   1:  PR[GP1:91,2] = PR[GP1:90,2] + -5.537;
   1:L PR[91] R[100]mm/sec CNT100;
   1:  PR[GP1:91,1] = PR[GP1:90,1] + 5.978;
   1:  PR[GP1:91,2] = PR[GP1:90,2] + -5.676;
   1:L PR[91] R[100]mm/sec CNT100;
   1:  PR[GP1:91,1] = PR[GP1:90,1] + 6.769;
   1:  PR[GP1:91,2] = PR[GP1:90,2] + -8.850;
   1:L PR[91] R[100]mm/sec CNT100;
   1:  PR[GP1:91,1] = PR[GP1:90,1] + 8.278;
   1:  PR[GP1:91,2] = PR[GP1:90,2] + -13.405;
   1:L PR[91] R[100]mm/sec CNT100;
   1:  PR[GP1:91,1] = PR[GP1:90,1] + 9.857;
   1:  PR[GP1:91,2] = PR[GP1:90,2] + -16.839;
   1:L PR[91] R[100]mm/sec CNT100;
   1:  PR[GP1:91,1] = PR[GP1:90,1] + 12.060;
   1:  PR[GP1:91,2] = PR[GP1:90,2] + -19.938;
   1:L PR[91] R[100]mm/sec CNT100;
   1:  PR[GP1:91,1] = PR[GP1:90,1] + 14.845;
   1:  PR[GP1:91,2] = PR[GP1:90,2] + -23.585;
   1:L PR[91] R[100]mm/sec CNT100;
   1:  PR[GP1:91,1] = PR[GP1:90,1] + 17.678;
   1:  PR[GP1:91,2] = PR[GP1:90,2] + -26.309;
   1:L PR[91] R[100]mm/sec CNT100;
   1:  PR[GP1:91,1] = PR[GP1:90,1] + 21.008;
   1:  PR[GP1:91,2] = PR[GP1:90,2] + -28.486;
   1:L PR[91] R[100]mm/sec CNT100;
   1:  PR[GP1:91,1] = PR[GP1:90,1] + 24.610;
   1:  PR[GP1:91,2] = PR[GP1:90,2] + -30.876;
   1:L PR[91] R[100]mm/sec CNT100;
   1:  PR[GP1:91,1] = PR[GP1:90,1] + 28.410;
   1:  PR[GP1:91,2] = PR[GP1:90,2] + -32.447;
   1:L PR[91] R[100]mm/sec CNT100;
   1:  PR[GP1:91,1] = PR[GP1:90,1] + 32.508;
   1:  PR[GP1:91,2] = PR[GP1:90,2] + -33.300;
   1:L PR[91] R[100]mm/sec CNT100;
   1:  PR[GP1:91,1] = PR[GP1:90,1] + 36.402;
   1:  PR[GP1:91,2] = PR[GP1:90,2] + -34.309;
   1:L PR[91] R[100]mm/sec CNT100;
   1:  PR[GP1:91,1] = PR[GP1:90,1] + 40.720;
   1:  PR[GP1:91,2] = PR[GP1:90,2] + -34.387;
   1:L PR[91] R[100]mm/sec CNT100;
   1:  PR[GP1:91,1] = PR[GP1:90,1] + 44.267;
   1:  PR[GP1:91,2] = PR[GP1:90,2] + -34.120;
   1:L PR[91] R[100]mm/sec CNT100;
   1:  PR[GP1:91,1] = PR[GP1:90,1] + 48.703;
   1:  PR[GP1:91,2] = PR[GP1:90,2] + -33.364;
   1:L PR[91] R[100]mm/sec CNT100;
   1:  PR[GP1:91,1] = PR[GP1:90,1] + 52.933;
   1:  PR[GP1:91,2] = PR[GP1:90,2] + -31.793;
   1:L PR[91] R[100]mm/sec CNT100;
   1:  PR[GP1:91,1] = PR[GP1:90,1] + 55.982;
   1:  PR[GP1:91,2] = PR[GP1:90,2] + -30.480;
   1:L PR[91] R[100]mm/sec CNT100;
   1:  PR[GP1:91,1] = PR[GP1:90,1] + 59.937;
   1:  PR[GP1:91,2] = PR[GP1:90,2] + -28.095;
   1:L PR[91] R[100]mm/sec CNT100;
   1:  PR[GP1:91,1] = PR[GP1:90,1] + 63.408;
   1:  PR[GP1:91,2] = PR[GP1:90,2] + -24.992;
   1:L PR[91] R[100]mm/sec CNT100;
   1:  PR[GP1:91,1] = PR[GP1:90,1] + 65.721;
   1:  PR[GP1:91,2] = PR[GP1:90,2] + -22.883;
   1:L PR[91] R[100]mm/sec CNT100;
   1:  PR[GP1:91,1] = PR[GP1:90,1] + 68.581;
   1:  PR[GP1:91,2] = PR[GP1:90,2] + -19.155;
   1:L PR[91] R[100]mm/sec CNT100;
   1:  PR[GP1:91,1] = PR[GP1:90,1] + 70.726;
   1:  PR[GP1:91,2] = PR[GP1:90,2] + -14.904;
   1:L PR[91] R[100]mm/sec CNT100;
   1:  PR[GP1:91,1] = PR[GP1:90,1] + 72.157;
   1:  PR[GP1:91,2] = PR[GP1:90,2] + -12.278;
   1:L PR[91] R[100]mm/sec CNT100;
   1:  PR[GP1:91,1] = PR[GP1:90,1] + 73.469;
   1:  PR[GP1:91,2] = PR[GP1:90,2] + -7.723;
   1:L PR[91] R[100]mm/sec CNT100;
   1:  PR[GP1:91,1] = PR[GP1:90,1] + 73.920;
   1:  PR[GP1:91,2] = PR[GP1:90,2] + -2.915;
   1:L PR[91] R[100]mm/sec CNT100;
   1:  PR[GP1:91,1] = PR[GP1:90,1] + 74.398;
   1:  PR[GP1:91,2] = PR[GP1:90,2] + -0.050;
   1:L PR[91] R[100]mm/sec CNT100;
   1:  PR[GP1:91,1] = PR[GP1:90,1] + 73.947;
   1:  PR[GP1:91,2] = PR[GP1:90,2] + 4.751;
   1:L PR[91] R[100]mm/sec CNT100;
   1:  PR[GP1:91,1] = PR[GP1:90,1] + 73.475;
   1:  PR[GP1:91,2] = PR[GP1:90,2] + 7.557;
   1:L PR[91] R[100]mm/sec CNT100;
   1:  PR[GP1:91,1] = PR[GP1:90,1] + 72.155;
   1:  PR[GP1:91,2] = PR[GP1:90,2] + 12.144;
   1:L PR[91] R[100]mm/sec CNT100;
   1:  PR[GP1:91,1] = PR[GP1:90,1] + 69.993;
   1:  PR[GP1:91,2] = PR[GP1:90,2] + 16.426;
   1:L PR[91] R[100]mm/sec CNT100;
   1:  PR[GP1:91,1] = PR[GP1:90,1] + 68.587;
   1:  PR[GP1:91,2] = PR[GP1:90,2] + 19.003;
   1:L PR[91] R[100]mm/sec CNT100;
   1:  PR[GP1:91,1] = PR[GP1:90,1] + 65.723;
   1:  PR[GP1:91,2] = PR[GP1:90,2] + 22.736;
   1:L PR[91] R[100]mm/sec CNT100;
   1:  PR[GP1:91,1] = PR[GP1:90,1] + 62.179;
   1:  PR[GP1:91,2] = PR[GP1:90,2] + 25.906;
   1:L PR[91] R[100]mm/sec CNT100;
   1:  PR[GP1:91,1] = PR[GP1:90,1] + 59.934;
   1:  PR[GP1:91,2] = PR[GP1:90,2] + 27.953;
   1:L PR[91] R[100]mm/sec CNT100;
   1:  PR[GP1:91,1] = PR[GP1:90,1] + 55.996;
   1:  PR[GP1:91,2] = PR[GP1:90,2] + 30.328;
   1:L PR[91] R[100]mm/sec CNT100;
   1:  PR[GP1:91,1] = PR[GP1:90,1] + 51.614;
   1:  PR[GP1:91,2] = PR[GP1:90,2] + 31.956;
   1:L PR[91] R[100]mm/sec CNT100;
   1:  PR[GP1:91,1] = PR[GP1:90,1] + 48.687;
   1:  PR[GP1:91,2] = PR[GP1:90,2] + 33.223;
   1:L PR[91] R[100]mm/sec CNT100;
   1:  PR[GP1:91,1] = PR[GP1:90,1] + 44.267;
   1:  PR[GP1:91,2] = PR[GP1:90,2] + 33.976;
   1:L PR[91] R[100]mm/sec CNT100;
   1:  PR[GP1:91,1] = PR[GP1:90,1] + 40.720;
   1:  PR[GP1:91,2] = PR[GP1:90,2] + 34.243;
   1:L PR[91] R[100]mm/sec CNT100;
   1:  PR[GP1:91,1] = PR[GP1:90,1] + 36.387;
   1:  PR[GP1:91,2] = PR[GP1:90,2] + 34.164;
   1:L PR[91] R[100]mm/sec CNT100;
   1:  PR[GP1:91,1] = PR[GP1:90,1] + 32.132;
   1:  PR[GP1:91,2] = PR[GP1:90,2] + 33.279;
   1:L PR[91] R[100]mm/sec CNT100;
   1:  PR[GP1:91,1] = PR[GP1:90,1] + 28.424;
   1:  PR[GP1:91,2] = PR[GP1:90,2] + 32.309;
   1:L PR[91] R[100]mm/sec CNT100;
   1:  PR[GP1:91,1] = PR[GP1:90,1] + 24.608;
   1:  PR[GP1:91,2] = PR[GP1:90,2] + 30.731;
   1:L PR[91] R[100]mm/sec CNT100;
   1:  PR[GP1:91,1] = PR[GP1:90,1] + 21.119;
   1:  PR[GP1:91,2] = PR[GP1:90,2] + 28.450;
   1:L PR[91] R[100]mm/sec CNT100;
   1:  PR[GP1:91,1] = PR[GP1:90,1] + 17.679;
   1:  PR[GP1:91,2] = PR[GP1:90,2] + 26.167;
   1:L PR[91] R[100]mm/sec CNT100;
   1:  PR[GP1:91,1] = PR[GP1:90,1] + 14.852;
   1:  PR[GP1:91,2] = PR[GP1:90,2] + 23.448;
   1:L PR[91] R[100]mm/sec CNT100;
   1:  PR[GP1:91,1] = PR[GP1:90,1] + 12.542;
   1:  PR[GP1:91,2] = PR[GP1:90,2] + 20.198;
   1:L PR[91] R[100]mm/sec CNT100;
   1:  PR[GP1:91,1] = PR[GP1:90,1] + 9.853;
   1:  PR[GP1:91,2] = PR[GP1:90,2] + 16.685;
   1:L PR[91] R[100]mm/sec CNT100;
   1:  PR[GP1:91,1] = PR[GP1:90,1] + 8.278;
   1:  PR[GP1:91,2] = PR[GP1:90,2] + 13.260;
   1:L PR[91] R[100]mm/sec CNT100;
   1:  PR[GP1:91,1] = PR[GP1:90,1] + 6.768;
   1:  PR[GP1:91,2] = PR[GP1:90,2] + 8.705;
   1:L PR[91] R[100]mm/sec CNT100;
   1:  PR[GP1:91,1] = PR[GP1:90,1] + 5.978;
   1:  PR[GP1:91,2] = PR[GP1:90,2] + 5.528;
   1:L PR[91] R[100]mm/sec CNT100;
   1:  PR[GP1:91,1] = PR[GP1:90,1] + 6.180;
   1:  PR[GP1:91,2] = PR[GP1:90,2] + 5.411;
   1:L PR[91] R[100]mm/sec CNT100;
   1:  PR[GP1:91,1] = PR[GP1:90,1] + 5.396;
   1:  PR[GP1:91,2] = PR[GP1:90,2] + 3.903;
   1:L PR[91] R[100]mm/sec CNT100;
   1:  PR[GP1:91,1] = PR[GP1:90,1] + 4.420;
   1:  PR[GP1:91,2] = PR[GP1:90,2] + 2.139;
   1:L PR[91] R[100]mm/sec CNT100;
   1:  PR[GP1:91,1] = PR[GP1:90,1] + 4.020;
   1:  PR[GP1:91,2] = PR[GP1:90,2] + 1.705;
   1:L PR[91] R[100]mm/sec CNT100;
   1:  PR[GP1:91,1] = PR[GP1:90,1] + 3.424;
   1:  PR[GP1:91,2] = PR[GP1:90,2] + 1.294;
   1:L PR[91] R[100]mm/sec CNT100;
   1:  PR[GP1:91,1] = PR[GP1:90,1] + 1.586;
   1:  PR[GP1:91,2] = PR[GP1:90,2] + 0.613;
   1:L PR[91] R[100]mm/sec CNT100;
   1:  PR[GP1:91,1] = PR[GP1:90,1] + 0.518;
   1:  PR[GP1:91,2] = PR[GP1:90,2] + 0.328;
   1:L PR[91] R[100]mm/sec CNT100;
   1:  PR[GP1:91,1] = PR[GP1:90,1] + -0.343;
   1:L PR[91] R[100]mm/sec CNT100;
   1:  ! -- Layer/Ebene 19 -- !;
   1:  PR[91] = PR[90];
   1:  PR[GP1:91,1] = PR[GP1:90,1] + -1.554;
   1:  PR[GP1:91,2] = PR[GP1:90,2] + 0.832;
   1:  PR[GP1:91,3] = PR[GP1:90,3] + 11.895;
   1:L PR[91] R[100]mm/sec CNT100;
   1:  PR[GP1:91,1] = PR[GP1:90,1] + -1.689;
   1:  PR[GP1:91,2] = PR[GP1:90,2] + 0.838;
   1:L PR[91] R[100]mm/sec CNT100;
   1:  PR[GP1:91,1] = PR[GP1:90,1] + -3.762;
   1:  PR[GP1:91,2] = PR[GP1:90,2] + 1.659;
   1:L PR[91] R[100]mm/sec CNT100;
   1:  PR[GP1:91,1] = PR[GP1:90,1] + -4.583;
   1:  PR[GP1:91,2] = PR[GP1:90,2] + 3.142;
   1:L PR[91] R[100]mm/sec CNT100;
   1:  PR[GP1:91,1] = PR[GP1:90,1] + -4.620;
   1:  PR[GP1:91,2] = PR[GP1:90,2] + 3.175;
   1:L PR[91] R[100]mm/sec CNT100;
   1:  PR[GP1:91,1] = PR[GP1:90,1] + -5.982;
   1:  PR[GP1:91,2] = PR[GP1:90,2] + 5.397;
   1:L PR[91] R[100]mm/sec CNT100;
   1:  PR[GP1:91,1] = PR[GP1:90,1] + -5.721;
   1:  PR[GP1:91,2] = PR[GP1:90,2] + 5.544;
   1:L PR[91] R[100]mm/sec CNT100;
   1:  PR[GP1:91,1] = PR[GP1:90,1] + -6.373;
   1:  PR[GP1:91,2] = PR[GP1:90,2] + 8.163;
   1:L PR[91] R[100]mm/sec CNT100;
   1:  PR[GP1:91,1] = PR[GP1:90,1] + -8.196;
   1:  PR[GP1:91,2] = PR[GP1:90,2] + 13.665;
   1:L PR[91] R[100]mm/sec CNT100;
   1:  PR[GP1:91,1] = PR[GP1:90,1] + -9.548;
   1:  PR[GP1:91,2] = PR[GP1:90,2] + 16.603;
   1:L PR[91] R[100]mm/sec CNT100;
   1:  PR[GP1:91,1] = PR[GP1:90,1] + -11.435;
   1:  PR[GP1:91,2] = PR[GP1:90,2] + 19.258;
   1:L PR[91] R[100]mm/sec CNT100;
   1:  PR[GP1:91,1] = PR[GP1:90,1] + -14.796;
   1:  PR[GP1:91,2] = PR[GP1:90,2] + 23.659;
   1:L PR[91] R[100]mm/sec CNT100;
   1:  PR[GP1:91,1] = PR[GP1:90,1] + -17.260;
   1:  PR[GP1:91,2] = PR[GP1:90,2] + 26.029;
   1:L PR[91] R[100]mm/sec CNT100;
   1:  PR[GP1:91,1] = PR[GP1:90,1] + -20.162;
   1:  PR[GP1:91,2] = PR[GP1:90,2] + 27.926;
   1:L PR[91] R[100]mm/sec CNT100;
   1:  PR[GP1:91,1] = PR[GP1:90,1] + -24.511;
   1:  PR[GP1:91,2] = PR[GP1:90,2] + 30.810;
   1:L PR[91] R[100]mm/sec CNT100;
   1:  PR[GP1:91,1] = PR[GP1:90,1] + -27.875;
   1:  PR[GP1:91,2] = PR[GP1:90,2] + 32.201;
   1:L PR[91] R[100]mm/sec CNT100;
   1:  PR[GP1:91,1] = PR[GP1:90,1] + -31.510;
   1:  PR[GP1:91,2] = PR[GP1:90,2] + 32.958;
   1:L PR[91] R[100]mm/sec CNT100;
   1:  PR[GP1:91,1] = PR[GP1:90,1] + -36.213;
   1:  PR[GP1:91,2] = PR[GP1:90,2] + 34.175;
   1:L PR[91] R[100]mm/sec CNT100;
   1:  PR[GP1:91,1] = PR[GP1:90,1] + -40.098;
   1:  PR[GP1:91,2] = PR[GP1:90,2] + 34.246;
   1:L PR[91] R[100]mm/sec CNT100;
   1:  PR[GP1:91,1] = PR[GP1:90,1] + -44.382;
   1:  PR[GP1:91,2] = PR[GP1:90,2] + 33.924;
   1:L PR[91] R[100]mm/sec CNT100;
   1:  PR[GP1:91,1] = PR[GP1:90,1] + -48.425;
   1:  PR[GP1:91,2] = PR[GP1:90,2] + 33.235;
   1:L PR[91] R[100]mm/sec CNT100;
   1:  PR[GP1:91,1] = PR[GP1:90,1] + -52.280;
   1:  PR[GP1:91,2] = PR[GP1:90,2] + 31.803;
   1:L PR[91] R[100]mm/sec CNT100;
   1:  PR[GP1:91,1] = PR[GP1:90,1] + -55.965;
   1:  PR[GP1:91,2] = PR[GP1:90,2] + 30.215;
   1:L PR[91] R[100]mm/sec CNT100;
   1:  PR[GP1:91,1] = PR[GP1:90,1] + -59.600;
   1:  PR[GP1:91,2] = PR[GP1:90,2] + 28.023;
   1:L PR[91] R[100]mm/sec CNT100;
   1:  PR[GP1:91,1] = PR[GP1:90,1] + -62.793;
   1:  PR[GP1:91,2] = PR[GP1:90,2] + 25.168;
   1:L PR[91] R[100]mm/sec CNT100;
   1:  PR[GP1:91,1] = PR[GP1:90,1] + -65.589;
   1:  PR[GP1:91,2] = PR[GP1:90,2] + 22.620;
   1:L PR[91] R[100]mm/sec CNT100;
   1:  PR[GP1:91,1] = PR[GP1:90,1] + -68.234;
   1:  PR[GP1:91,2] = PR[GP1:90,2] + 19.173;
   1:L PR[91] R[100]mm/sec CNT100;
   1:  PR[GP1:91,1] = PR[GP1:90,1] + -70.219;
   1:  PR[GP1:91,2] = PR[GP1:90,2] + 15.237;
   1:L PR[91] R[100]mm/sec CNT100;
   1:  PR[GP1:91,1] = PR[GP1:90,1] + -71.949;
   1:  PR[GP1:91,2] = PR[GP1:90,2] + 12.062;
   1:L PR[91] R[100]mm/sec CNT100;
   1:  PR[GP1:91,1] = PR[GP1:90,1] + -73.167;
   1:  PR[GP1:91,2] = PR[GP1:90,2] + 7.835;
   1:L PR[91] R[100]mm/sec CNT100;
   1:  PR[GP1:91,1] = PR[GP1:90,1] + -73.586;
   1:  PR[GP1:91,2] = PR[GP1:90,2] + 3.368;
   1:L PR[91] R[100]mm/sec CNT100;
   1:  PR[GP1:91,1] = PR[GP1:90,1] + -74.163;
   1:  PR[GP1:91,2] = PR[GP1:90,2] + -0.094;
   1:L PR[91] R[100]mm/sec CNT100;
   1:  PR[GP1:91,1] = PR[GP1:90,1] + -73.744;
   1:  PR[GP1:91,2] = PR[GP1:90,2] + -4.567;
   1:L PR[91] R[100]mm/sec CNT100;
   1:  PR[GP1:91,1] = PR[GP1:90,1] + -73.173;
   1:  PR[GP1:91,2] = PR[GP1:90,2] + -7.957;
   1:L PR[91] R[100]mm/sec CNT100;
   1:  PR[GP1:91,1] = PR[GP1:90,1] + -71.947;
   1:  PR[GP1:91,2] = PR[GP1:90,2] + -12.215;
   1:L PR[91] R[100]mm/sec CNT100;
   1:  PR[GP1:91,1] = PR[GP1:90,1] + -69.940;
   1:  PR[GP1:91,2] = PR[GP1:90,2] + -16.192;
   1:L PR[91] R[100]mm/sec CNT100;
   1:  PR[GP1:91,1] = PR[GP1:90,1] + -68.239;
   1:  PR[GP1:91,2] = PR[GP1:90,2] + -19.309;
   1:L PR[91] R[100]mm/sec CNT100;
   1:  PR[GP1:91,1] = PR[GP1:90,1] + -65.591;
   1:  PR[GP1:91,2] = PR[GP1:90,2] + -22.762;
   1:L PR[91] R[100]mm/sec CNT100;
   1:  PR[GP1:91,1] = PR[GP1:90,1] + -62.310;
   1:  PR[GP1:91,2] = PR[GP1:90,2] + -25.696;
   1:L PR[91] R[100]mm/sec CNT100;
   1:  PR[GP1:91,1] = PR[GP1:90,1] + -59.598;
   1:  PR[GP1:91,2] = PR[GP1:90,2] + -28.169;
   1:L PR[91] R[100]mm/sec CNT100;
   1:  PR[GP1:91,1] = PR[GP1:90,1] + -55.978;
   1:  PR[GP1:91,2] = PR[GP1:90,2] + -30.352;
   1:L PR[91] R[100]mm/sec CNT100;
   1:  PR[GP1:91,1] = PR[GP1:90,1] + -51.945;
   1:  PR[GP1:91,2] = PR[GP1:90,2] + -31.850;
   1:L PR[91] R[100]mm/sec CNT100;
   1:  PR[GP1:91,1] = PR[GP1:90,1] + -48.409;
   1:  PR[GP1:91,2] = PR[GP1:90,2] + -33.382;
   1:L PR[91] R[100]mm/sec CNT100;
   1:  PR[GP1:91,1] = PR[GP1:90,1] + -44.383;
   1:  PR[GP1:91,2] = PR[GP1:90,2] + -34.068;
   1:L PR[91] R[100]mm/sec CNT100;
   1:  PR[GP1:91,1] = PR[GP1:90,1] + -40.098;
   1:  PR[GP1:91,2] = PR[GP1:90,2] + -34.390;
   1:L PR[91] R[100]mm/sec CNT100;
   1:  PR[GP1:91,1] = PR[GP1:90,1] + -36.198;
   1:  PR[GP1:91,2] = PR[GP1:90,2] + -34.319;
   1:L PR[91] R[100]mm/sec CNT100;
   1:  PR[GP1:91,1] = PR[GP1:90,1] + -32.367;
   1:  PR[GP1:91,2] = PR[GP1:90,2] + -33.522;
   1:L PR[91] R[100]mm/sec CNT100;
   1:  PR[GP1:91,1] = PR[GP1:90,1] + -27.889;
   1:  PR[GP1:91,2] = PR[GP1:90,2] + -32.351;
   1:L PR[91] R[100]mm/sec CNT100;
   1:  PR[GP1:91,1] = PR[GP1:90,1] + -24.509;
   1:  PR[GP1:91,2] = PR[GP1:90,2] + -30.954;
   1:L PR[91] R[100]mm/sec CNT100;
   1:  PR[GP1:91,1] = PR[GP1:90,1] + -21.416;
   1:  PR[GP1:91,2] = PR[GP1:90,2] + -28.932;
   1:L PR[91] R[100]mm/sec CNT100;
   1:  PR[GP1:91,1] = PR[GP1:90,1] + -17.262;
   1:  PR[GP1:91,2] = PR[GP1:90,2] + -26.174;
   1:L PR[91] R[100]mm/sec CNT100;
   1:  PR[GP1:91,1] = PR[GP1:90,1] + -14.804;
   1:  PR[GP1:91,2] = PR[GP1:90,2] + -23.810;
   1:L PR[91] R[100]mm/sec CNT100;
   1:  PR[GP1:91,1] = PR[GP1:90,1] + -12.790;
   1:  PR[GP1:91,2] = PR[GP1:90,2] + -20.977;
   1:L PR[91] R[100]mm/sec CNT100;
   1:  PR[GP1:91,1] = PR[GP1:90,1] + -9.543;
   1:  PR[GP1:91,2] = PR[GP1:90,2] + -16.738;
   1:L PR[91] R[100]mm/sec CNT100;
   1:  PR[GP1:91,1] = PR[GP1:90,1] + -8.197;
   1:  PR[GP1:91,2] = PR[GP1:90,2] + -13.809;
   1:L PR[91] R[100]mm/sec CNT100;
   1:  PR[GP1:91,1] = PR[GP1:90,1] + -6.374;
   1:  PR[GP1:91,2] = PR[GP1:90,2] + -8.308;
   1:L PR[91] R[100]mm/sec CNT100;
   1:  PR[GP1:91,1] = PR[GP1:90,1] + -5.720;
   1:  PR[GP1:91,2] = PR[GP1:90,2] + -5.683;
   1:L PR[91] R[100]mm/sec CNT100;
   1:  PR[GP1:91,1] = PR[GP1:90,1] + -5.941;
   1:  PR[GP1:91,2] = PR[GP1:90,2] + -5.553;
   1:L PR[91] R[100]mm/sec CNT100;
   1:  PR[GP1:91,1] = PR[GP1:90,1] + -5.053;
   1:  PR[GP1:91,2] = PR[GP1:90,2] + -3.844;
   1:L PR[91] R[100]mm/sec CNT100;
   1:  PR[GP1:91,1] = PR[GP1:90,1] + -4.229;
   1:  PR[GP1:91,2] = PR[GP1:90,2] + -2.356;
   1:L PR[91] R[100]mm/sec CNT100;
   1:  PR[GP1:91,1] = PR[GP1:90,1] + -3.767;
   1:  PR[GP1:91,2] = PR[GP1:90,2] + -1.854;
   1:L PR[91] R[100]mm/sec CNT100;
   1:  PR[GP1:91,1] = PR[GP1:90,1] + -3.073;
   1:  PR[GP1:91,2] = PR[GP1:90,2] + -1.376;
   1:L PR[91] R[100]mm/sec CNT100;
   1:  PR[GP1:91,1] = PR[GP1:90,1] + -1.546;
   1:  PR[GP1:91,2] = PR[GP1:90,2] + -0.809;
   1:L PR[91] R[100]mm/sec CNT100;
   1:  PR[GP1:91,1] = PR[GP1:90,1] + -0.580;
   1:  PR[GP1:91,2] = PR[GP1:90,2] + -0.552;
   1:L PR[91] R[100]mm/sec CNT100;
   1:  PR[GP1:91,1] = PR[GP1:90,1] + -0.247;
   1:  PR[GP1:91,2] = PR[GP1:90,2] + -0.472;
   1:L PR[91] R[100]mm/sec CNT100;
   1:  PR[GP1:91,1] = PR[GP1:90,1] + 0.503;
   1:L PR[91] R[100]mm/sec CNT100;
   1:  PR[GP1:91,1] = PR[GP1:90,1] + 1.767;
   1:  PR[GP1:91,2] = PR[GP1:90,2] + -0.976;
   1:L PR[91] R[100]mm/sec CNT100;
   1:  PR[GP1:91,1] = PR[GP1:90,1] + 1.902;
   1:  PR[GP1:91,2] = PR[GP1:90,2] + -0.982;
   1:L PR[91] R[100]mm/sec CNT100;
   1:  PR[GP1:91,1] = PR[GP1:90,1] + 3.975;
   1:  PR[GP1:91,2] = PR[GP1:90,2] + -1.803;
   1:L PR[91] R[100]mm/sec CNT100;
   1:  PR[GP1:91,1] = PR[GP1:90,1] + 4.797;
   1:  PR[GP1:91,2] = PR[GP1:90,2] + -3.286;
   1:L PR[91] R[100]mm/sec CNT100;
   1:  PR[GP1:91,1] = PR[GP1:90,1] + 4.833;
   1:  PR[GP1:91,2] = PR[GP1:90,2] + -3.320;
   1:L PR[91] R[100]mm/sec CNT100;
   1:  PR[GP1:91,1] = PR[GP1:90,1] + 6.194;
   1:  PR[GP1:91,2] = PR[GP1:90,2] + -5.539;
   1:L PR[91] R[100]mm/sec CNT100;
   1:  PR[GP1:91,1] = PR[GP1:90,1] + 5.934;
   1:  PR[GP1:91,2] = PR[GP1:90,2] + -5.688;
   1:L PR[91] R[100]mm/sec CNT100;
   1:  PR[GP1:91,1] = PR[GP1:90,1] + 6.587;
   1:  PR[GP1:91,2] = PR[GP1:90,2] + -8.309;
   1:L PR[91] R[100]mm/sec CNT100;
   1:  PR[GP1:91,1] = PR[GP1:90,1] + 8.409;
   1:  PR[GP1:91,2] = PR[GP1:90,2] + -13.806;
   1:L PR[91] R[100]mm/sec CNT100;
   1:  PR[GP1:91,1] = PR[GP1:90,1] + 9.760;
   1:  PR[GP1:91,2] = PR[GP1:90,2] + -16.745;
   1:L PR[91] R[100]mm/sec CNT100;
   1:  PR[GP1:91,1] = PR[GP1:90,1] + 11.647;
   1:  PR[GP1:91,2] = PR[GP1:90,2] + -19.400;
   1:L PR[91] R[100]mm/sec CNT100;
   1:  PR[GP1:91,1] = PR[GP1:90,1] + 15.009;
   1:  PR[GP1:91,2] = PR[GP1:90,2] + -23.802;
   1:L PR[91] R[100]mm/sec CNT100;
   1:  PR[GP1:91,1] = PR[GP1:90,1] + 17.473;
   1:  PR[GP1:91,2] = PR[GP1:90,2] + -26.172;
   1:L PR[91] R[100]mm/sec CNT100;
   1:  PR[GP1:91,1] = PR[GP1:90,1] + 20.374;
   1:  PR[GP1:91,2] = PR[GP1:90,2] + -28.069;
   1:L PR[91] R[100]mm/sec CNT100;
   1:  PR[GP1:91,1] = PR[GP1:90,1] + 24.723;
   1:  PR[GP1:91,2] = PR[GP1:90,2] + -30.954;
   1:L PR[91] R[100]mm/sec CNT100;
   1:  PR[GP1:91,1] = PR[GP1:90,1] + 28.087;
   1:  PR[GP1:91,2] = PR[GP1:90,2] + -32.345;
   1:L PR[91] R[100]mm/sec CNT100;
   1:  PR[GP1:91,1] = PR[GP1:90,1] + 31.723;
   1:  PR[GP1:91,2] = PR[GP1:90,2] + -33.101;
   1:L PR[91] R[100]mm/sec CNT100;
   1:  PR[GP1:91,1] = PR[GP1:90,1] + 36.425;
   1:  PR[GP1:91,2] = PR[GP1:90,2] + -34.319;
   1:L PR[91] R[100]mm/sec CNT100;
   1:  PR[GP1:91,1] = PR[GP1:90,1] + 40.310;
   1:  PR[GP1:91,2] = PR[GP1:90,2] + -34.390;
   1:L PR[91] R[100]mm/sec CNT100;
   1:  PR[GP1:91,1] = PR[GP1:90,1] + 44.595;
   1:  PR[GP1:91,2] = PR[GP1:90,2] + -34.068;
   1:L PR[91] R[100]mm/sec CNT100;
   1:  PR[GP1:91,1] = PR[GP1:90,1] + 48.637;
   1:  PR[GP1:91,2] = PR[GP1:90,2] + -33.379;
   1:L PR[91] R[100]mm/sec CNT100;
   1:  PR[GP1:91,1] = PR[GP1:90,1] + 52.493;
   1:  PR[GP1:91,2] = PR[GP1:90,2] + -31.947;
   1:L PR[91] R[100]mm/sec CNT100;
   1:  PR[GP1:91,1] = PR[GP1:90,1] + 56.178;
   1:  PR[GP1:91,2] = PR[GP1:90,2] + -30.360;
   1:L PR[91] R[100]mm/sec CNT100;
   1:  PR[GP1:91,1] = PR[GP1:90,1] + 59.813;
   1:  PR[GP1:91,2] = PR[GP1:90,2] + -28.168;
   1:L PR[91] R[100]mm/sec CNT100;
   1:  PR[GP1:91,1] = PR[GP1:90,1] + 63.006;
   1:  PR[GP1:91,2] = PR[GP1:90,2] + -25.312;
   1:L PR[91] R[100]mm/sec CNT100;
   1:  PR[GP1:91,1] = PR[GP1:90,1] + 65.802;
   1:  PR[GP1:91,2] = PR[GP1:90,2] + -22.764;
   1:L PR[91] R[100]mm/sec CNT100;
   1:  PR[GP1:91,1] = PR[GP1:90,1] + 68.447;
   1:  PR[GP1:91,2] = PR[GP1:90,2] + -19.316;
   1:L PR[91] R[100]mm/sec CNT100;
   1:  PR[GP1:91,1] = PR[GP1:90,1] + 70.433;
   1:  PR[GP1:91,2] = PR[GP1:90,2] + -15.381;
   1:L PR[91] R[100]mm/sec CNT100;
   1:  PR[GP1:91,1] = PR[GP1:90,1] + 72.163;
   1:  PR[GP1:91,2] = PR[GP1:90,2] + -12.207;
   1:L PR[91] R[100]mm/sec CNT100;
   1:  PR[GP1:91,1] = PR[GP1:90,1] + 73.380;
   1:  PR[GP1:91,2] = PR[GP1:90,2] + -7.980;
   1:L PR[91] R[100]mm/sec CNT100;
   1:  PR[GP1:91,1] = PR[GP1:90,1] + 73.799;
   1:  PR[GP1:91,2] = PR[GP1:90,2] + -3.513;
   1:L PR[91] R[100]mm/sec CNT100;
   1:  PR[GP1:91,1] = PR[GP1:90,1] + 74.376;
   1:  PR[GP1:91,2] = PR[GP1:90,2] + -0.050;
   1:L PR[91] R[100]mm/sec CNT100;
   1:  PR[GP1:91,1] = PR[GP1:90,1] + 73.957;
   1:  PR[GP1:91,2] = PR[GP1:90,2] + 4.423;
   1:L PR[91] R[100]mm/sec CNT100;
   1:  PR[GP1:91,1] = PR[GP1:90,1] + 73.386;
   1:  PR[GP1:91,2] = PR[GP1:90,2] + 7.815;
   1:L PR[91] R[100]mm/sec CNT100;
   1:  PR[GP1:91,1] = PR[GP1:90,1] + 72.160;
   1:  PR[GP1:91,2] = PR[GP1:90,2] + 12.072;
   1:L PR[91] R[100]mm/sec CNT100;
   1:  PR[GP1:91,1] = PR[GP1:90,1] + 70.153;
   1:  PR[GP1:91,2] = PR[GP1:90,2] + 16.050;
   1:L PR[91] R[100]mm/sec CNT100;
   1:  PR[GP1:91,1] = PR[GP1:90,1] + 68.453;
   1:  PR[GP1:91,2] = PR[GP1:90,2] + 19.164;
   1:L PR[91] R[100]mm/sec CNT100;
   1:  PR[GP1:91,1] = PR[GP1:90,1] + 65.804;
   1:  PR[GP1:91,2] = PR[GP1:90,2] + 22.617;
   1:L PR[91] R[100]mm/sec CNT100;
   1:  PR[GP1:91,1] = PR[GP1:90,1] + 62.523;
   1:  PR[GP1:91,2] = PR[GP1:90,2] + 25.551;
   1:L PR[91] R[100]mm/sec CNT100;
   1:  PR[GP1:91,1] = PR[GP1:90,1] + 59.810;
   1:  PR[GP1:91,2] = PR[GP1:90,2] + 28.025;
   1:L PR[91] R[100]mm/sec CNT100;
   1:  PR[GP1:91,1] = PR[GP1:90,1] + 56.191;
   1:  PR[GP1:91,2] = PR[GP1:90,2] + 30.208;
   1:L PR[91] R[100]mm/sec CNT100;
   1:  PR[GP1:91,1] = PR[GP1:90,1] + 52.158;
   1:  PR[GP1:91,2] = PR[GP1:90,2] + 31.706;
   1:L PR[91] R[100]mm/sec CNT100;
   1:  PR[GP1:91,1] = PR[GP1:90,1] + 48.621;
   1:  PR[GP1:91,2] = PR[GP1:90,2] + 33.238;
   1:L PR[91] R[100]mm/sec CNT100;
   1:  PR[GP1:91,1] = PR[GP1:90,1] + 44.595;
   1:  PR[GP1:91,2] = PR[GP1:90,2] + 33.924;
   1:L PR[91] R[100]mm/sec CNT100;
   1:  PR[GP1:91,1] = PR[GP1:90,1] + 40.310;
   1:  PR[GP1:91,2] = PR[GP1:90,2] + 34.246;
   1:L PR[91] R[100]mm/sec CNT100;
   1:  PR[GP1:91,1] = PR[GP1:90,1] + 36.410;
   1:  PR[GP1:91,2] = PR[GP1:90,2] + 34.175;
   1:L PR[91] R[100]mm/sec CNT100;
   1:  PR[GP1:91,1] = PR[GP1:90,1] + 32.579;
   1:  PR[GP1:91,2] = PR[GP1:90,2] + 33.378;
   1:L PR[91] R[100]mm/sec CNT100;
   1:  PR[GP1:91,1] = PR[GP1:90,1] + 28.102;
   1:  PR[GP1:91,2] = PR[GP1:90,2] + 32.207;
   1:L PR[91] R[100]mm/sec CNT100;
   1:  PR[GP1:91,1] = PR[GP1:90,1] + 24.721;
   1:  PR[GP1:91,2] = PR[GP1:90,2] + 30.809;
   1:L PR[91] R[100]mm/sec CNT100;
   1:  PR[GP1:91,1] = PR[GP1:90,1] + 21.627;
   1:  PR[GP1:91,2] = PR[GP1:90,2] + 28.786;
   1:L PR[91] R[100]mm/sec CNT100;
   1:  PR[GP1:91,1] = PR[GP1:90,1] + 17.474;
   1:  PR[GP1:91,2] = PR[GP1:90,2] + 26.030;
   1:L PR[91] R[100]mm/sec CNT100;
   1:  PR[GP1:91,1] = PR[GP1:90,1] + 15.016;
   1:  PR[GP1:91,2] = PR[GP1:90,2] + 23.665;
   1:L PR[91] R[100]mm/sec CNT100;
   1:  PR[GP1:91,1] = PR[GP1:90,1] + 13.003;
   1:  PR[GP1:91,2] = PR[GP1:90,2] + 20.833;
   1:L PR[91] R[100]mm/sec CNT100;
   1:  PR[GP1:91,1] = PR[GP1:90,1] + 9.756;
   1:  PR[GP1:91,2] = PR[GP1:90,2] + 16.591;
   1:L PR[91] R[100]mm/sec CNT100;
   1:  PR[GP1:91,1] = PR[GP1:90,1] + 8.409;
   1:  PR[GP1:91,2] = PR[GP1:90,2] + 13.662;
   1:L PR[91] R[100]mm/sec CNT100;
   1:  PR[GP1:91,1] = PR[GP1:90,1] + 6.586;
   1:  PR[GP1:91,2] = PR[GP1:90,2] + 8.163;
   1:L PR[91] R[100]mm/sec CNT100;
   1:  PR[GP1:91,1] = PR[GP1:90,1] + 5.933;
   1:  PR[GP1:91,2] = PR[GP1:90,2] + 5.540;
   1:L PR[91] R[100]mm/sec CNT100;
   1:  PR[GP1:91,1] = PR[GP1:90,1] + 6.155;
   1:  PR[GP1:91,2] = PR[GP1:90,2] + 5.412;
   1:L PR[91] R[100]mm/sec CNT100;
   1:  PR[GP1:91,1] = PR[GP1:90,1] + 5.266;
   1:  PR[GP1:91,2] = PR[GP1:90,2] + 3.700;
   1:L PR[91] R[100]mm/sec CNT100;
   1:  PR[GP1:91,1] = PR[GP1:90,1] + 4.442;
   1:  PR[GP1:91,2] = PR[GP1:90,2] + 2.212;
   1:L PR[91] R[100]mm/sec CNT100;
   1:  PR[GP1:91,1] = PR[GP1:90,1] + 3.980;
   1:  PR[GP1:91,2] = PR[GP1:90,2] + 1.710;
   1:L PR[91] R[100]mm/sec CNT100;
   1:  PR[GP1:91,1] = PR[GP1:90,1] + 3.286;
   1:  PR[GP1:91,2] = PR[GP1:90,2] + 1.232;
   1:L PR[91] R[100]mm/sec CNT100;
   1:  PR[GP1:91,1] = PR[GP1:90,1] + 1.759;
   1:  PR[GP1:91,2] = PR[GP1:90,2] + 0.665;
   1:L PR[91] R[100]mm/sec CNT100;
   1:  PR[GP1:91,1] = PR[GP1:90,1] + 0.790;
   1:  PR[GP1:91,2] = PR[GP1:90,2] + 0.407;
   1:L PR[91] R[100]mm/sec CNT100;
   1:  PR[GP1:91,1] = PR[GP1:90,1] + 0.461;
   1:  PR[GP1:91,2] = PR[GP1:90,2] + 0.328;
   1:L PR[91] R[100]mm/sec CNT100;
   1:  PR[GP1:91,1] = PR[GP1:90,1] + -0.290;
   1:L PR[91] R[100]mm/sec CNT100;
   1:  ! -- Layer/Ebene 20 -- !;
   1:  PR[91] = PR[90];
   1:  PR[GP1:91,1] = PR[GP1:90,1] + -1.184;
   1:  PR[GP1:91,2] = PR[GP1:90,2] + 0.712;
   1:  PR[GP1:91,3] = PR[GP1:90,3] + 12.505;
   1:L PR[91] R[100]mm/sec CNT100;
   1:  PR[GP1:91,1] = PR[GP1:90,1] + -1.342;
   1:  PR[GP1:91,2] = PR[GP1:90,2] + 0.719;
   1:L PR[91] R[100]mm/sec CNT100;
   1:  PR[GP1:91,1] = PR[GP1:90,1] + -3.717;
   1:  PR[GP1:91,2] = PR[GP1:90,2] + 1.659;
   1:L PR[91] R[100]mm/sec CNT100;
   1:  PR[GP1:91,1] = PR[GP1:90,1] + -4.382;
   1:  PR[GP1:91,2] = PR[GP1:90,2] + 2.860;
   1:L PR[91] R[100]mm/sec CNT100;
   1:  PR[GP1:91,1] = PR[GP1:90,1] + -4.426;
   1:  PR[GP1:91,2] = PR[GP1:90,2] + 2.900;
   1:L PR[91] R[100]mm/sec CNT100;
   1:  PR[GP1:91,1] = PR[GP1:90,1] + -5.256;
   1:  PR[GP1:91,2] = PR[GP1:90,2] + 4.249;
   1:L PR[91] R[100]mm/sec CNT100;
   1:  PR[GP1:91,1] = PR[GP1:90,1] + -5.662;
   1:  PR[GP1:91,2] = PR[GP1:90,2] + 4.998;
   1:L PR[91] R[100]mm/sec CNT100;
   1:  PR[GP1:91,1] = PR[GP1:90,1] + -5.720;
   1:  PR[GP1:91,2] = PR[GP1:90,2] + 5.532;
   1:L PR[91] R[100]mm/sec CNT100;
   1:  PR[GP1:91,1] = PR[GP1:90,1] + -5.677;
   1:  PR[GP1:91,2] = PR[GP1:90,2] + 5.556;
   1:L PR[91] R[100]mm/sec CNT100;
   1:  PR[GP1:91,1] = PR[GP1:90,1] + -6.191;
   1:  PR[GP1:91,2] = PR[GP1:90,2] + 7.621;
   1:L PR[91] R[100]mm/sec CNT100;
   1:  PR[GP1:91,1] = PR[GP1:90,1] + -8.327;
   1:  PR[GP1:91,2] = PR[GP1:90,2] + 14.067;
   1:L PR[91] R[100]mm/sec CNT100;
   1:  PR[GP1:91,1] = PR[GP1:90,1] + -9.451;
   1:  PR[GP1:91,2] = PR[GP1:90,2] + 16.510;
   1:L PR[91] R[100]mm/sec CNT100;
   1:  PR[GP1:91,1] = PR[GP1:90,1] + -11.022;
   1:  PR[GP1:91,2] = PR[GP1:90,2] + 18.721;
   1:L PR[91] R[100]mm/sec CNT100;
   1:  PR[GP1:91,1] = PR[GP1:90,1] + -14.960;
   1:  PR[GP1:91,2] = PR[GP1:90,2] + 23.876;
   1:L PR[91] R[100]mm/sec CNT100;
   1:  PR[GP1:91,1] = PR[GP1:90,1] + -17.055;
   1:  PR[GP1:91,2] = PR[GP1:90,2] + 25.892;
   1:L PR[91] R[100]mm/sec CNT100;
   1:  PR[GP1:91,1] = PR[GP1:90,1] + -19.529;
   1:  PR[GP1:91,2] = PR[GP1:90,2] + 27.508;
   1:L PR[91] R[100]mm/sec CNT100;
   1:  PR[GP1:91,1] = PR[GP1:90,1] + -24.625;
   1:  PR[GP1:91,2] = PR[GP1:90,2] + 30.889;
   1:L PR[91] R[100]mm/sec CNT100;
   1:  PR[GP1:91,1] = PR[GP1:90,1] + -27.552;
   1:  PR[GP1:91,2] = PR[GP1:90,2] + 32.099;
   1:L PR[91] R[100]mm/sec CNT100;
   1:  PR[GP1:91,1] = PR[GP1:90,1] + -30.725;
   1:  PR[GP1:91,2] = PR[GP1:90,2] + 32.759;
   1:L PR[91] R[100]mm/sec CNT100;
   1:  PR[GP1:91,1] = PR[GP1:90,1] + -36.236;
   1:  PR[GP1:91,2] = PR[GP1:90,2] + 34.186;
   1:L PR[91] R[100]mm/sec CNT100;
   1:  PR[GP1:91,1] = PR[GP1:90,1] + -39.688;
   1:  PR[GP1:91,2] = PR[GP1:90,2] + 34.249;
   1:L PR[91] R[100]mm/sec CNT100;
   1:  PR[GP1:91,1] = PR[GP1:90,1] + -44.710;
   1:  PR[GP1:91,2] = PR[GP1:90,2] + 33.871;
   1:L PR[91] R[100]mm/sec CNT100;
   1:  PR[GP1:91,1] = PR[GP1:90,1] + -48.359;
   1:  PR[GP1:91,2] = PR[GP1:90,2] + 33.249;
   1:L PR[91] R[100]mm/sec CNT100;
   1:  PR[GP1:91,1] = PR[GP1:90,1] + -51.841;
   1:  PR[GP1:91,2] = PR[GP1:90,2] + 31.956;
   1:L PR[91] R[100]mm/sec CNT100;
   1:  PR[GP1:91,1] = PR[GP1:90,1] + -56.160;
   1:  PR[GP1:91,2] = PR[GP1:90,2] + 30.096;
   1:L PR[91] R[100]mm/sec CNT100;
   1:  PR[GP1:91,1] = PR[GP1:90,1] + -59.477;
   1:  PR[GP1:91,2] = PR[GP1:90,2] + 28.095;
   1:L PR[91] R[100]mm/sec CNT100;
   1:  PR[GP1:91,1] = PR[GP1:90,1] + -62.393;
   1:  PR[GP1:91,2] = PR[GP1:90,2] + 25.488;
   1:L PR[91] R[100]mm/sec CNT100;
   1:  PR[GP1:91,1] = PR[GP1:90,1] + -65.670;
   1:  PR[GP1:91,2] = PR[GP1:90,2] + 22.501;
   1:L PR[91] R[100]mm/sec CNT100;
   1:  PR[GP1:91,1] = PR[GP1:90,1] + -68.100;
   1:  PR[GP1:91,2] = PR[GP1:90,2] + 19.334;
   1:L PR[91] R[100]mm/sec CNT100;
   1:  PR[GP1:91,1] = PR[GP1:90,1] + -69.926;
   1:  PR[GP1:91,2] = PR[GP1:90,2] + 15.714;
   1:L PR[91] R[100]mm/sec CNT100;
   1:  PR[GP1:91,1] = PR[GP1:90,1] + -71.955;
   1:  PR[GP1:91,2] = PR[GP1:90,2] + 11.990;
   1:L PR[91] R[100]mm/sec CNT100;
   1:  PR[GP1:91,1] = PR[GP1:90,1] + -73.078;
   1:  PR[GP1:91,2] = PR[GP1:90,2] + 8.092;
   1:L PR[91] R[100]mm/sec CNT100;
   1:  PR[GP1:91,1] = PR[GP1:90,1] + -73.465;
   1:  PR[GP1:91,2] = PR[GP1:90,2] + 3.965;
   1:L PR[91] R[100]mm/sec CNT100;
   1:  PR[GP1:91,1] = PR[GP1:90,1] + -74.142;
   1:  PR[GP1:91,2] = PR[GP1:90,2] + -0.094;
   1:L PR[91] R[100]mm/sec CNT100;
   1:  PR[GP1:91,1] = PR[GP1:90,1] + -73.753;
   1:  PR[GP1:91,2] = PR[GP1:90,2] + -4.239;
   1:L PR[91] R[100]mm/sec CNT100;
   1:  PR[GP1:91,1] = PR[GP1:90,1] + -73.084;
   1:  PR[GP1:91,2] = PR[GP1:90,2] + -8.214;
   1:L PR[91] R[100]mm/sec CNT100;
   1:  PR[GP1:91,1] = PR[GP1:90,1] + -71.952;
   1:  PR[GP1:91,2] = PR[GP1:90,2] + -12.144;
   1:L PR[91] R[100]mm/sec CNT100;
   1:  PR[GP1:91,1] = PR[GP1:90,1] + -70.099;
   1:  PR[GP1:91,2] = PR[GP1:90,2] + -15.816;
   1:L PR[91] R[100]mm/sec CNT100;
   1:  PR[GP1:91,1] = PR[GP1:90,1] + -68.106;
   1:  PR[GP1:91,2] = PR[GP1:90,2] + -19.470;
   1:L PR[91] R[100]mm/sec CNT100;
   1:  PR[GP1:91,1] = PR[GP1:90,1] + -65.672;
   1:  PR[GP1:91,2] = PR[GP1:90,2] + -22.643;
   1:L PR[91] R[100]mm/sec CNT100;
   1:  PR[GP1:91,1] = PR[GP1:90,1] + -62.654;
   1:  PR[GP1:91,2] = PR[GP1:90,2] + -25.341;
   1:L PR[91] R[100]mm/sec CNT100;
   1:  PR[GP1:91,1] = PR[GP1:90,1] + -59.474;
   1:  PR[GP1:91,2] = PR[GP1:90,2] + -28.241;
   1:L PR[91] R[100]mm/sec CNT100;
   1:  PR[GP1:91,1] = PR[GP1:90,1] + -56.173;
   1:  PR[GP1:91,2] = PR[GP1:90,2] + -30.232;
   1:L PR[91] R[100]mm/sec CNT100;
   1:  PR[GP1:91,1] = PR[GP1:90,1] + -52.489;
   1:  PR[GP1:91,2] = PR[GP1:90,2] + -31.600;
   1:L PR[91] R[100]mm/sec CNT100;
   1:  PR[GP1:91,1] = PR[GP1:90,1] + -48.343;
   1:  PR[GP1:91,2] = PR[GP1:90,2] + -33.396;
   1:L PR[91] R[100]mm/sec CNT100;
   1:  PR[GP1:91,1] = PR[GP1:90,1] + -44.710;
   1:  PR[GP1:91,2] = PR[GP1:90,2] + -34.015;
   1:L PR[91] R[100]mm/sec CNT100;
   1:  PR[GP1:91,1] = PR[GP1:90,1] + -39.688;
   1:  PR[GP1:91,2] = PR[GP1:90,2] + -34.393;
   1:L PR[91] R[100]mm/sec CNT100;
   1:  PR[GP1:91,1] = PR[GP1:90,1] + -36.221;
   1:  PR[GP1:91,2] = PR[GP1:90,2] + -34.330;
   1:L PR[91] R[100]mm/sec CNT100;
   1:  PR[GP1:91,1] = PR[GP1:90,1] + -32.814;
   1:  PR[GP1:91,2] = PR[GP1:90,2] + -33.621;
   1:L PR[91] R[100]mm/sec CNT100;
   1:  PR[GP1:91,1] = PR[GP1:90,1] + -27.567;
   1:  PR[GP1:91,2] = PR[GP1:90,2] + -32.249;
   1:L PR[91] R[100]mm/sec CNT100;
   1:  PR[GP1:91,1] = PR[GP1:90,1] + -24.623;
   1:  PR[GP1:91,2] = PR[GP1:90,2] + -31.032;
   1:L PR[91] R[100]mm/sec CNT100;
   1:  PR[GP1:91,1] = PR[GP1:90,1] + -21.924;
   1:  PR[GP1:91,2] = PR[GP1:90,2] + -29.268;
   1:L PR[91] R[100]mm/sec CNT100;
   1:  PR[GP1:91,1] = PR[GP1:90,1] + -17.057;
   1:  PR[GP1:91,2] = PR[GP1:90,2] + -26.037;
   1:L PR[91] R[100]mm/sec CNT100;
   1:  PR[GP1:91,1] = PR[GP1:90,1] + -14.968;
   1:  PR[GP1:91,2] = PR[GP1:90,2] + -24.027;
   1:L PR[91] R[100]mm/sec CNT100;
   1:  PR[GP1:91,1] = PR[GP1:90,1] + -13.251;
   1:  PR[GP1:91,2] = PR[GP1:90,2] + -21.612;
   1:L PR[91] R[100]mm/sec CNT100;
   1:  PR[GP1:91,1] = PR[GP1:90,1] + -9.446;
   1:  PR[GP1:91,2] = PR[GP1:90,2] + -16.644;
   1:L PR[91] R[100]mm/sec CNT100;
   1:  PR[GP1:91,1] = PR[GP1:90,1] + -8.327;
   1:  PR[GP1:91,2] = PR[GP1:90,2] + -14.211;
   1:L PR[91] R[100]mm/sec CNT100;
   1:  PR[GP1:91,1] = PR[GP1:90,1] + -6.192;
   1:  PR[GP1:91,2] = PR[GP1:90,2] + -7.767;
   1:L PR[91] R[100]mm/sec CNT100;
   1:  PR[GP1:91,1] = PR[GP1:90,1] + -5.676;
   1:  PR[GP1:91,2] = PR[GP1:90,2] + -5.694;
   1:L PR[91] R[100]mm/sec CNT100;
   1:  PR[GP1:91,1] = PR[GP1:90,1] + -5.721;
   1:  PR[GP1:91,2] = PR[GP1:90,2] + -5.668;
   1:L PR[91] R[100]mm/sec CNT100;
   1:  PR[GP1:91,1] = PR[GP1:90,1] + -5.667;
   1:  PR[GP1:91,2] = PR[GP1:90,2] + -5.172;
   1:L PR[91] R[100]mm/sec CNT100;
   1:  PR[GP1:91,1] = PR[GP1:90,1] + -5.450;
   1:  PR[GP1:91,2] = PR[GP1:90,2] + -4.655;
   1:L PR[91] R[100]mm/sec CNT100;
   1:  PR[GP1:91,1] = PR[GP1:90,1] + -4.923;
   1:  PR[GP1:91,2] = PR[GP1:90,2] + -3.641;
   1:L PR[91] R[100]mm/sec CNT100;
   1:  PR[GP1:91,1] = PR[GP1:90,1] + -4.252;
   1:  PR[GP1:91,2] = PR[GP1:90,2] + -2.429;
   1:L PR[91] R[100]mm/sec CNT100;
   1:  PR[GP1:91,1] = PR[GP1:90,1] + -3.727;
   1:  PR[GP1:91,2] = PR[GP1:90,2] + -1.859;
   1:L PR[91] R[100]mm/sec CNT100;
   1:  PR[GP1:91,1] = PR[GP1:90,1] + -2.935;
   1:  PR[GP1:91,2] = PR[GP1:90,2] + -1.313;
   1:L PR[91] R[100]mm/sec CNT100;
   1:  PR[GP1:91,1] = PR[GP1:90,1] + -1.718;
   1:  PR[GP1:91,2] = PR[GP1:90,2] + -0.862;
   1:L PR[91] R[100]mm/sec CNT100;
   1:  PR[GP1:91,1] = PR[GP1:90,1] + -0.955;
   1:  PR[GP1:91,2] = PR[GP1:90,2] + -0.658;
   1:L PR[91] R[100]mm/sec CNT100;
   1:  PR[GP1:91,1] = PR[GP1:90,1] + -0.179;
   1:  PR[GP1:91,2] = PR[GP1:90,2] + -0.472;
   1:L PR[91] R[100]mm/sec CNT100;
   1:  PR[GP1:91,1] = PR[GP1:90,1] + 0.435;
   1:L PR[91] R[100]mm/sec CNT100;
   1:  PR[GP1:91,1] = PR[GP1:90,1] + 1.397;
   1:  PR[GP1:91,2] = PR[GP1:90,2] + -0.856;
   1:L PR[91] R[100]mm/sec CNT100;
   1:  PR[GP1:91,1] = PR[GP1:90,1] + 1.555;
   1:  PR[GP1:91,2] = PR[GP1:90,2] + -0.863;
   1:L PR[91] R[100]mm/sec CNT100;
   1:  PR[GP1:91,1] = PR[GP1:90,1] + 3.930;
   1:  PR[GP1:91,2] = PR[GP1:90,2] + -1.803;
   1:L PR[91] R[100]mm/sec CNT100;
   1:  PR[GP1:91,1] = PR[GP1:90,1] + 4.596;
   1:  PR[GP1:91,2] = PR[GP1:90,2] + -3.004;
   1:L PR[91] R[100]mm/sec CNT100;
   1:  PR[GP1:91,1] = PR[GP1:90,1] + 4.640;
   1:  PR[GP1:91,2] = PR[GP1:90,2] + -3.045;
   1:L PR[91] R[100]mm/sec CNT100;
   1:  PR[GP1:91,1] = PR[GP1:90,1] + 5.469;
   1:  PR[GP1:91,2] = PR[GP1:90,2] + -4.393;
   1:L PR[91] R[100]mm/sec CNT100;
   1:  PR[GP1:91,1] = PR[GP1:90,1] + 5.875;
   1:  PR[GP1:91,2] = PR[GP1:90,2] + -5.142;
   1:L PR[91] R[100]mm/sec CNT100;
   1:  PR[GP1:91,1] = PR[GP1:90,1] + 5.933;
   1:  PR[GP1:91,2] = PR[GP1:90,2] + -5.675;
   1:L PR[91] R[100]mm/sec CNT100;
   1:  PR[GP1:91,1] = PR[GP1:90,1] + 5.890;
   1:  PR[GP1:91,2] = PR[GP1:90,2] + -5.700;
   1:L PR[91] R[100]mm/sec CNT100;
   1:  PR[GP1:91,1] = PR[GP1:90,1] + 6.405;
   1:  PR[GP1:91,2] = PR[GP1:90,2] + -7.767;
   1:L PR[91] R[100]mm/sec CNT100;
   1:  PR[GP1:91,1] = PR[GP1:90,1] + 8.540;
   1:  PR[GP1:91,2] = PR[GP1:90,2] + -14.208;
   1:L PR[91] R[100]mm/sec CNT100;
   1:  PR[GP1:91,1] = PR[GP1:90,1] + 9.663;
   1:  PR[GP1:91,2] = PR[GP1:90,2] + -16.651;
   1:L PR[91] R[100]mm/sec CNT100;
   1:  PR[GP1:91,1] = PR[GP1:90,1] + 11.234;
   1:  PR[GP1:91,2] = PR[GP1:90,2] + -18.862;
   1:L PR[91] R[100]mm/sec CNT100;
   1:  PR[GP1:91,1] = PR[GP1:90,1] + 15.172;
   1:  PR[GP1:91,2] = PR[GP1:90,2] + -24.020;
   1:L PR[91] R[100]mm/sec CNT100;
   1:  PR[GP1:91,1] = PR[GP1:90,1] + 17.268;
   1:  PR[GP1:91,2] = PR[GP1:90,2] + -26.035;
   1:L PR[91] R[100]mm/sec CNT100;
   1:  PR[GP1:91,1] = PR[GP1:90,1] + 19.741;
   1:  PR[GP1:91,2] = PR[GP1:90,2] + -27.652;
   1:L PR[91] R[100]mm/sec CNT100;
   1:  PR[GP1:91,1] = PR[GP1:90,1] + 24.837;
   1:  PR[GP1:91,2] = PR[GP1:90,2] + -31.032;
   1:L PR[91] R[100]mm/sec CNT100;
   1:  PR[GP1:91,1] = PR[GP1:90,1] + 27.764;
   1:  PR[GP1:91,2] = PR[GP1:90,2] + -32.243;
   1:L PR[91] R[100]mm/sec CNT100;
   1:  PR[GP1:91,1] = PR[GP1:90,1] + 30.938;
   1:  PR[GP1:91,2] = PR[GP1:90,2] + -32.903;
   1:L PR[91] R[100]mm/sec CNT100;
   1:  PR[GP1:91,1] = PR[GP1:90,1] + 36.448;
   1:  PR[GP1:91,2] = PR[GP1:90,2] + -34.330;
   1:L PR[91] R[100]mm/sec CNT100;
   1:  PR[GP1:91,1] = PR[GP1:90,1] + 39.900;
   1:  PR[GP1:91,2] = PR[GP1:90,2] + -34.393;
   1:L PR[91] R[100]mm/sec CNT100;
   1:  PR[GP1:91,1] = PR[GP1:90,1] + 44.923;
   1:  PR[GP1:91,2] = PR[GP1:90,2] + -34.015;
   1:L PR[91] R[100]mm/sec CNT100;
   1:  PR[GP1:91,1] = PR[GP1:90,1] + 48.572;
   1:  PR[GP1:91,2] = PR[GP1:90,2] + -33.393;
   1:L PR[91] R[100]mm/sec CNT100;
   1:  PR[GP1:91,1] = PR[GP1:90,1] + 52.053;
   1:  PR[GP1:91,2] = PR[GP1:90,2] + -32.100;
   1:L PR[91] R[100]mm/sec CNT100;
   1:  PR[GP1:91,1] = PR[GP1:90,1] + 56.373;
   1:  PR[GP1:91,2] = PR[GP1:90,2] + -30.240;
   1:L PR[91] R[100]mm/sec CNT100;
   1:  PR[GP1:91,1] = PR[GP1:90,1] + 59.689;
   1:  PR[GP1:91,2] = PR[GP1:90,2] + -28.240;
   1:L PR[91] R[100]mm/sec CNT100;
   1:  PR[GP1:91,1] = PR[GP1:90,1] + 62.605;
   1:  PR[GP1:91,2] = PR[GP1:90,2] + -25.633;
   1:L PR[91] R[100]mm/sec CNT100;
   1:  PR[GP1:91,1] = PR[GP1:90,1] + 65.883;
   1:  PR[GP1:91,2] = PR[GP1:90,2] + -22.645;
   1:L PR[91] R[100]mm/sec CNT100;
   1:  PR[GP1:91,1] = PR[GP1:90,1] + 68.313;
   1:  PR[GP1:91,2] = PR[GP1:90,2] + -19.477;
   1:L PR[91] R[100]mm/sec CNT100;
   1:  PR[GP1:91,1] = PR[GP1:90,1] + 70.139;
   1:  PR[GP1:91,2] = PR[GP1:90,2] + -15.857;
   1:L PR[91] R[100]mm/sec CNT100;
   1:  PR[GP1:91,1] = PR[GP1:90,1] + 72.168;
   1:  PR[GP1:91,2] = PR[GP1:90,2] + -12.136;
   1:L PR[91] R[100]mm/sec CNT100;
   1:  PR[GP1:91,1] = PR[GP1:90,1] + 73.291;
   1:  PR[GP1:91,2] = PR[GP1:90,2] + -8.237;
   1:L PR[91] R[100]mm/sec CNT100;
   1:  PR[GP1:91,1] = PR[GP1:90,1] + 73.678;
   1:  PR[GP1:91,2] = PR[GP1:90,2] + -4.111;
   1:L PR[91] R[100]mm/sec CNT100;
   1:  PR[GP1:91,1] = PR[GP1:90,1] + 74.355;
   1:  PR[GP1:91,2] = PR[GP1:90,2] + -0.050;
   1:L PR[91] R[100]mm/sec CNT100;
   1:  PR[GP1:91,1] = PR[GP1:90,1] + 73.966;
   1:  PR[GP1:91,2] = PR[GP1:90,2] + 4.095;
   1:L PR[91] R[100]mm/sec CNT100;
   1:  PR[GP1:91,1] = PR[GP1:90,1] + 73.297;
   1:  PR[GP1:91,2] = PR[GP1:90,2] + 8.072;
   1:L PR[91] R[100]mm/sec CNT100;
   1:  PR[GP1:91,1] = PR[GP1:90,1] + 72.165;
   1:  PR[GP1:91,2] = PR[GP1:90,2] + 12.001;
   1:L PR[91] R[100]mm/sec CNT100;
   1:  PR[GP1:91,1] = PR[GP1:90,1] + 70.312;
   1:  PR[GP1:91,2] = PR[GP1:90,2] + 15.673;
   1:L PR[91] R[100]mm/sec CNT100;
   1:  PR[GP1:91,1] = PR[GP1:90,1] + 68.319;
   1:  PR[GP1:91,2] = PR[GP1:90,2] + 19.325;
   1:L PR[91] R[100]mm/sec CNT100;
   1:  PR[GP1:91,1] = PR[GP1:90,1] + 65.885;
   1:  PR[GP1:91,2] = PR[GP1:90,2] + 22.498;
   1:L PR[91] R[100]mm/sec CNT100;
   1:  PR[GP1:91,1] = PR[GP1:90,1] + 62.867;
   1:  PR[GP1:91,2] = PR[GP1:90,2] + 25.197;
   1:L PR[91] R[100]mm/sec CNT100;
   1:  PR[GP1:91,1] = PR[GP1:90,1] + 59.687;
   1:  PR[GP1:91,2] = PR[GP1:90,2] + 28.098;
   1:L PR[91] R[100]mm/sec CNT100;
   1:  PR[GP1:91,1] = PR[GP1:90,1] + 56.386;
   1:  PR[GP1:91,2] = PR[GP1:90,2] + 30.088;
   1:L PR[91] R[100]mm/sec CNT100;
   1:  PR[GP1:91,1] = PR[GP1:90,1] + 52.702;
   1:  PR[GP1:91,2] = PR[GP1:90,2] + 31.457;
   1:L PR[91] R[100]mm/sec CNT100;
   1:  PR[GP1:91,1] = PR[GP1:90,1] + 48.556;
   1:  PR[GP1:91,2] = PR[GP1:90,2] + 33.252;
   1:L PR[91] R[100]mm/sec CNT100;
   1:  PR[GP1:91,1] = PR[GP1:90,1] + 44.923;
   1:  PR[GP1:91,2] = PR[GP1:90,2] + 33.871;
   1:L PR[91] R[100]mm/sec CNT100;
   1:  PR[GP1:91,1] = PR[GP1:90,1] + 39.900;
   1:  PR[GP1:91,2] = PR[GP1:90,2] + 34.249;
   1:L PR[91] R[100]mm/sec CNT100;
   1:  PR[GP1:91,1] = PR[GP1:90,1] + 36.434;
   1:  PR[GP1:91,2] = PR[GP1:90,2] + 34.186;
   1:L PR[91] R[100]mm/sec CNT100;
   1:  PR[GP1:91,1] = PR[GP1:90,1] + 33.027;
   1:  PR[GP1:91,2] = PR[GP1:90,2] + 33.477;
   1:L PR[91] R[100]mm/sec CNT100;
   1:  PR[GP1:91,1] = PR[GP1:90,1] + 27.779;
   1:  PR[GP1:91,2] = PR[GP1:90,2] + 32.104;
   1:L PR[91] R[100]mm/sec CNT100;
   1:  PR[GP1:91,1] = PR[GP1:90,1] + 24.835;
   1:  PR[GP1:91,2] = PR[GP1:90,2] + 30.887;
   1:L PR[91] R[100]mm/sec CNT100;
   1:  PR[GP1:91,1] = PR[GP1:90,1] + 22.136;
   1:  PR[GP1:91,2] = PR[GP1:90,2] + 29.123;
   1:L PR[91] R[100]mm/sec CNT100;
   1:  PR[GP1:91,1] = PR[GP1:90,1] + 17.269;
   1:  PR[GP1:91,2] = PR[GP1:90,2] + 25.892;
   1:L PR[91] R[100]mm/sec CNT100;
   1:  PR[GP1:91,1] = PR[GP1:90,1] + 15.180;
   1:  PR[GP1:91,2] = PR[GP1:90,2] + 23.883;
   1:L PR[91] R[100]mm/sec CNT100;
   1:  PR[GP1:91,1] = PR[GP1:90,1] + 13.463;
   1:  PR[GP1:91,2] = PR[GP1:90,2] + 21.467;
   1:L PR[91] R[100]mm/sec CNT100;
   1:  PR[GP1:91,1] = PR[GP1:90,1] + 9.659;
   1:  PR[GP1:91,2] = PR[GP1:90,2] + 16.498;
   1:L PR[91] R[100]mm/sec CNT100;
   1:  PR[GP1:91,1] = PR[GP1:90,1] + 8.540;
   1:  PR[GP1:91,2] = PR[GP1:90,2] + 14.064;
   1:L PR[91] R[100]mm/sec CNT100;
   1:  PR[GP1:91,1] = PR[GP1:90,1] + 6.404;
   1:  PR[GP1:91,2] = PR[GP1:90,2] + 7.622;
   1:L PR[91] R[100]mm/sec CNT100;
   1:  PR[GP1:91,1] = PR[GP1:90,1] + 5.889;
   1:  PR[GP1:91,2] = PR[GP1:90,2] + 5.552;
   1:L PR[91] R[100]mm/sec CNT100;
   1:  PR[GP1:91,1] = PR[GP1:90,1] + 5.934;
   1:  PR[GP1:91,2] = PR[GP1:90,2] + 5.525;
   1:L PR[91] R[100]mm/sec CNT100;
   1:  PR[GP1:91,1] = PR[GP1:90,1] + 5.880;
   1:  PR[GP1:91,2] = PR[GP1:90,2] + 5.028;
   1:L PR[91] R[100]mm/sec CNT100;
   1:  PR[GP1:91,1] = PR[GP1:90,1] + 5.664;
   1:  PR[GP1:91,2] = PR[GP1:90,2] + 4.514;
   1:L PR[91] R[100]mm/sec CNT100;
   1:  PR[GP1:91,1] = PR[GP1:90,1] + 5.136;
   1:  PR[GP1:91,2] = PR[GP1:90,2] + 3.497;
   1:L PR[91] R[100]mm/sec CNT100;
   1:  PR[GP1:91,1] = PR[GP1:90,1] + 4.465;
   1:  PR[GP1:91,2] = PR[GP1:90,2] + 2.285;
   1:L PR[91] R[100]mm/sec CNT100;
   1:  PR[GP1:91,1] = PR[GP1:90,1] + 3.940;
   1:  PR[GP1:91,2] = PR[GP1:90,2] + 1.715;
   1:L PR[91] R[100]mm/sec CNT100;
   1:  PR[GP1:91,1] = PR[GP1:90,1] + 3.148;
   1:  PR[GP1:91,2] = PR[GP1:90,2] + 1.169;
   1:L PR[91] R[100]mm/sec CNT100;
   1:  PR[GP1:91,1] = PR[GP1:90,1] + 1.932;
   1:  PR[GP1:91,2] = PR[GP1:90,2] + 0.718;
   1:L PR[91] R[100]mm/sec CNT100;
   1:  PR[GP1:91,1] = PR[GP1:90,1] + 1.166;
   1:  PR[GP1:91,2] = PR[GP1:90,2] + 0.514;
   1:L PR[91] R[100]mm/sec CNT100;
   1:  PR[GP1:91,1] = PR[GP1:90,1] + 0.392;
   1:  PR[GP1:91,2] = PR[GP1:90,2] + 0.328;
   1:L PR[91] R[100]mm/sec CNT100;
   1:  PR[GP1:91,1] = PR[GP1:90,1] + -0.222;
   1:L PR[91] R[100]mm/sec CNT100;
   1:  ! -- Layer/Ebene 21 -- !;
   1:  PR[91] = PR[90];
   1:  PR[GP1:91,1] = PR[GP1:90,1] + -0.814;
   1:  PR[GP1:91,2] = PR[GP1:90,2] + 0.591;
   1:  PR[GP1:91,3] = PR[GP1:90,3] + 13.115;
   1:L PR[91] R[100]mm/sec CNT100;
   1:  PR[GP1:91,1] = PR[GP1:90,1] + -0.994;
   1:  PR[GP1:91,2] = PR[GP1:90,2] + 0.599;
   1:L PR[91] R[100]mm/sec CNT100;
   1:  PR[GP1:91,1] = PR[GP1:90,1] + -3.672;
   1:  PR[GP1:91,2] = PR[GP1:90,2] + 1.659;
   1:L PR[91] R[100]mm/sec CNT100;
   1:  PR[GP1:91,1] = PR[GP1:90,1] + -4.181;
   1:  PR[GP1:91,2] = PR[GP1:90,2] + 2.578;
   1:L PR[91] R[100]mm/sec CNT100;
   1:  PR[GP1:91,1] = PR[GP1:90,1] + -4.233;
   1:  PR[GP1:91,2] = PR[GP1:90,2] + 2.625;
   1:L PR[91] R[100]mm/sec CNT100;
   1:  PR[GP1:91,1] = PR[GP1:90,1] + -4.865;
   1:  PR[GP1:91,2] = PR[GP1:90,2] + 3.652;
   1:L PR[91] R[100]mm/sec CNT100;
   1:  PR[GP1:91,1] = PR[GP1:90,1] + -5.594;
   1:  PR[GP1:91,2] = PR[GP1:90,2] + 4.998;
   1:L PR[91] R[100]mm/sec CNT100;
   1:  PR[GP1:91,1] = PR[GP1:90,1] + -5.654;
   1:  PR[GP1:91,2] = PR[GP1:90,2] + 5.556;
   1:L PR[91] R[100]mm/sec CNT100;
   1:  PR[GP1:91,1] = PR[GP1:90,1] + -5.633;
   1:  PR[GP1:91,2] = PR[GP1:90,2] + 5.568;
   1:L PR[91] R[100]mm/sec CNT100;
   1:  PR[GP1:91,1] = PR[GP1:90,1] + -6.009;
   1:  PR[GP1:91,2] = PR[GP1:90,2] + 7.080;
   1:L PR[91] R[100]mm/sec CNT100;
   1:  PR[GP1:91,1] = PR[GP1:90,1] + -8.458;
   1:  PR[GP1:91,2] = PR[GP1:90,2] + 14.469;
   1:L PR[91] R[100]mm/sec CNT100;
   1:  PR[GP1:91,1] = PR[GP1:90,1] + -9.354;
   1:  PR[GP1:91,2] = PR[GP1:90,2] + 16.417;
   1:L PR[91] R[100]mm/sec CNT100;
   1:  PR[GP1:91,1] = PR[GP1:90,1] + -10.609;
   1:  PR[GP1:91,2] = PR[GP1:90,2] + 18.183;
   1:L PR[91] R[100]mm/sec CNT100;
   1:  PR[GP1:91,1] = PR[GP1:90,1] + -15.124;
   1:  PR[GP1:91,2] = PR[GP1:90,2] + 24.094;
   1:L PR[91] R[100]mm/sec CNT100;
   1:  PR[GP1:91,1] = PR[GP1:90,1] + -16.851;
   1:  PR[GP1:91,2] = PR[GP1:90,2] + 25.754;
   1:L PR[91] R[100]mm/sec CNT100;
   1:  PR[GP1:91,1] = PR[GP1:90,1] + -18.895;
   1:  PR[GP1:91,2] = PR[GP1:90,2] + 27.091;
   1:L PR[91] R[100]mm/sec CNT100;
   1:  PR[GP1:91,1] = PR[GP1:90,1] + -24.738;
   1:  PR[GP1:91,2] = PR[GP1:90,2] + 30.967;
   1:L PR[91] R[100]mm/sec CNT100;
   1:  PR[GP1:91,1] = PR[GP1:90,1] + -27.230;
   1:  PR[GP1:91,2] = PR[GP1:90,2] + 31.997;
   1:L PR[91] R[100]mm/sec CNT100;
   1:  PR[GP1:91,1] = PR[GP1:90,1] + -29.940;
   1:  PR[GP1:91,2] = PR[GP1:90,2] + 32.561;
   1:L PR[91] R[100]mm/sec CNT100;
   1:  PR[GP1:91,1] = PR[GP1:90,1] + -36.259;
   1:  PR[GP1:91,2] = PR[GP1:90,2] + 34.197;
   1:L PR[91] R[100]mm/sec CNT100;
   1:  PR[GP1:91,1] = PR[GP1:90,1] + -39.279;
   1:  PR[GP1:91,2] = PR[GP1:90,2] + 34.252;
   1:L PR[91] R[100]mm/sec CNT100;
   1:  PR[GP1:91,1] = PR[GP1:90,1] + -45.038;
   1:  PR[GP1:91,2] = PR[GP1:90,2] + 33.819;
   1:L PR[91] R[100]mm/sec CNT100;
   1:  PR[GP1:91,1] = PR[GP1:90,1] + -48.294;
   1:  PR[GP1:91,2] = PR[GP1:90,2] + 33.264;
   1:L PR[91] R[100]mm/sec CNT100;
   1:  PR[GP1:91,1] = PR[GP1:90,1] + -51.401;
   1:  PR[GP1:91,2] = PR[GP1:90,2] + 32.110;
   1:L PR[91] R[100]mm/sec CNT100;
   1:  PR[GP1:91,1] = PR[GP1:90,1] + -56.355;
   1:  PR[GP1:91,2] = PR[GP1:90,2] + 29.976;
   1:L PR[91] R[100]mm/sec CNT100;
   1:  PR[GP1:91,1] = PR[GP1:90,1] + -59.353;
   1:  PR[GP1:91,2] = PR[GP1:90,2] + 28.168;
   1:L PR[91] R[100]mm/sec CNT100;
   1:  PR[GP1:91,1] = PR[GP1:90,1] + -61.991;
   1:  PR[GP1:91,2] = PR[GP1:90,2] + 25.809;
   1:L PR[91] R[100]mm/sec CNT100;
   1:  PR[GP1:91,1] = PR[GP1:90,1] + -65.751;
   1:  PR[GP1:91,2] = PR[GP1:90,2] + 22.382;
   1:L PR[91] R[100]mm/sec CNT100;
   1:  PR[GP1:91,1] = PR[GP1:90,1] + -67.966;
   1:  PR[GP1:91,2] = PR[GP1:90,2] + 19.495;
   1:L PR[91] R[100]mm/sec CNT100;
   1:  PR[GP1:91,1] = PR[GP1:90,1] + -69.633;
   1:  PR[GP1:91,2] = PR[GP1:90,2] + 16.191;
   1:L PR[91] R[100]mm/sec CNT100;
   1:  PR[GP1:91,1] = PR[GP1:90,1] + -71.960;
   1:  PR[GP1:91,2] = PR[GP1:90,2] + 11.919;
   1:L PR[91] R[100]mm/sec CNT100;
   1:  PR[GP1:91,1] = PR[GP1:90,1] + -72.989;
   1:  PR[GP1:91,2] = PR[GP1:90,2] + 8.349;
   1:L PR[91] R[100]mm/sec CNT100;
   1:  PR[GP1:91,1] = PR[GP1:90,1] + -73.343;
   1:  PR[GP1:91,2] = PR[GP1:90,2] + 4.563;
   1:L PR[91] R[100]mm/sec CNT100;
   1:  PR[GP1:91,1] = PR[GP1:90,1] + -74.120;
   1:  PR[GP1:91,2] = PR[GP1:90,2] + -0.094;
   1:L PR[91] R[100]mm/sec CNT100;
   1:  PR[GP1:91,1] = PR[GP1:90,1] + -73.762;
   1:  PR[GP1:91,2] = PR[GP1:90,2] + -3.911;
   1:L PR[91] R[100]mm/sec CNT100;
   1:  PR[GP1:91,1] = PR[GP1:90,1] + -72.995;
   1:  PR[GP1:91,2] = PR[GP1:90,2] + -8.472;
   1:L PR[91] R[100]mm/sec CNT100;
   1:  PR[GP1:91,1] = PR[GP1:90,1] + -71.958;
   1:  PR[GP1:91,2] = PR[GP1:90,2] + -12.072;
   1:L PR[91] R[100]mm/sec CNT100;
   1:  PR[GP1:91,1] = PR[GP1:90,1] + -70.259;
   1:  PR[GP1:91,2] = PR[GP1:90,2] + -15.439;
   1:L PR[91] R[100]mm/sec CNT100;
   1:  PR[GP1:91,1] = PR[GP1:90,1] + -67.972;
   1:  PR[GP1:91,2] = PR[GP1:90,2] + -19.631;
   1:L PR[91] R[100]mm/sec CNT100;
   1:  PR[GP1:91,1] = PR[GP1:90,1] + -65.753;
   1:  PR[GP1:91,2] = PR[GP1:90,2] + -22.524;
   1:L PR[91] R[100]mm/sec CNT100;
   1:  PR[GP1:91,1] = PR[GP1:90,1] + -62.999;
   1:  PR[GP1:91,2] = PR[GP1:90,2] + -24.987;
   1:L PR[91] R[100]mm/sec CNT100;
   1:  PR[GP1:91,1] = PR[GP1:90,1] + -59.350;
   1:  PR[GP1:91,2] = PR[GP1:90,2] + -28.313;
   1:L PR[91] R[100]mm/sec CNT100;
   1:  PR[GP1:91,1] = PR[GP1:90,1] + -56.368;
   1:  PR[GP1:91,2] = PR[GP1:90,2] + -30.112;
   1:L PR[91] R[100]mm/sec CNT100;
   1:  PR[GP1:91,1] = PR[GP1:90,1] + -53.033;
   1:  PR[GP1:91,2] = PR[GP1:90,2] + -31.350;
   1:L PR[91] R[100]mm/sec CNT100;
   1:  PR[GP1:91,1] = PR[GP1:90,1] + -48.278;
   1:  PR[GP1:91,2] = PR[GP1:90,2] + -33.411;
   1:L PR[91] R[100]mm/sec CNT100;
   1:  PR[GP1:91,1] = PR[GP1:90,1] + -45.038;
   1:  PR[GP1:91,2] = PR[GP1:90,2] + -33.963;
   1:L PR[91] R[100]mm/sec CNT100;
   1:  PR[GP1:91,1] = PR[GP1:90,1] + -39.279;
   1:  PR[GP1:91,2] = PR[GP1:90,2] + -34.396;
   1:L PR[91] R[100]mm/sec CNT100;
   1:  PR[GP1:91,1] = PR[GP1:90,1] + -36.245;
   1:  PR[GP1:91,2] = PR[GP1:90,2] + -34.341;
   1:L PR[91] R[100]mm/sec CNT100;
   1:  PR[GP1:91,1] = PR[GP1:90,1] + -33.261;
   1:  PR[GP1:91,2] = PR[GP1:90,2] + -33.720;
   1:L PR[91] R[100]mm/sec CNT100;
   1:  PR[GP1:91,1] = PR[GP1:90,1] + -27.244;
   1:  PR[GP1:91,2] = PR[GP1:90,2] + -32.147;
   1:L PR[91] R[100]mm/sec CNT100;
   1:  PR[GP1:91,1] = PR[GP1:90,1] + -24.736;
   1:  PR[GP1:91,2] = PR[GP1:90,2] + -31.110;
   1:L PR[91] R[100]mm/sec CNT100;
   1:  PR[GP1:91,1] = PR[GP1:90,1] + -22.433;
   1:  PR[GP1:91,2] = PR[GP1:90,2] + -29.604;
   1:L PR[91] R[100]mm/sec CNT100;
   1:  PR[GP1:91,1] = PR[GP1:90,1] + -16.852;
   1:  PR[GP1:91,2] = PR[GP1:90,2] + -25.900;
   1:L PR[91] R[100]mm/sec CNT100;
   1:  PR[GP1:91,1] = PR[GP1:90,1] + -15.132;
   1:  PR[GP1:91,2] = PR[GP1:90,2] + -24.245;
   1:L PR[91] R[100]mm/sec CNT100;
   1:  PR[GP1:91,1] = PR[GP1:90,1] + -13.711;
   1:  PR[GP1:91,2] = PR[GP1:90,2] + -22.247;
   1:L PR[91] R[100]mm/sec CNT100;
   1:  PR[GP1:91,1] = PR[GP1:90,1] + -9.349;
   1:  PR[GP1:91,2] = PR[GP1:90,2] + -16.551;
   1:L PR[91] R[100]mm/sec CNT100;
   1:  PR[GP1:91,1] = PR[GP1:90,1] + -8.458;
   1:  PR[GP1:91,2] = PR[GP1:90,2] + -14.613;
   1:L PR[91] R[100]mm/sec CNT100;
   1:  PR[GP1:91,1] = PR[GP1:90,1] + -6.010;
   1:  PR[GP1:91,2] = PR[GP1:90,2] + -7.225;
   1:L PR[91] R[100]mm/sec CNT100;
   1:  PR[GP1:91,1] = PR[GP1:90,1] + -5.631;
   1:  PR[GP1:91,2] = PR[GP1:90,2] + -5.706;
   1:L PR[91] R[100]mm/sec CNT100;
   1:  PR[GP1:91,1] = PR[GP1:90,1] + -5.656;
   1:  PR[GP1:91,2] = PR[GP1:90,2] + -5.692;
   1:L PR[91] R[100]mm/sec CNT100;
   1:  PR[GP1:91,1] = PR[GP1:90,1] + -5.599;
   1:  PR[GP1:91,2] = PR[GP1:90,2] + -5.172;
   1:L PR[91] R[100]mm/sec CNT100;
   1:  PR[GP1:91,1] = PR[GP1:90,1] + -5.196;
   1:  PR[GP1:91,2] = PR[GP1:90,2] + -4.214;
   1:L PR[91] R[100]mm/sec CNT100;
   1:  PR[GP1:91,1] = PR[GP1:90,1] + -4.793;
   1:  PR[GP1:91,2] = PR[GP1:90,2] + -3.438;
   1:L PR[91] R[100]mm/sec CNT100;
   1:  PR[GP1:91,1] = PR[GP1:90,1] + -4.275;
   1:  PR[GP1:91,2] = PR[GP1:90,2] + -2.502;
   1:L PR[91] R[100]mm/sec CNT100;
   1:  PR[GP1:91,1] = PR[GP1:90,1] + -3.687;
   1:  PR[GP1:91,2] = PR[GP1:90,2] + -1.864;
   1:L PR[91] R[100]mm/sec CNT100;
   1:  PR[GP1:91,1] = PR[GP1:90,1] + -2.797;
   1:  PR[GP1:91,2] = PR[GP1:90,2] + -1.250;
   1:L PR[91] R[100]mm/sec CNT100;
   1:  PR[GP1:91,1] = PR[GP1:90,1] + -1.891;
   1:  PR[GP1:91,2] = PR[GP1:90,2] + -0.915;
   1:L PR[91] R[100]mm/sec CNT100;
   1:  PR[GP1:91,1] = PR[GP1:90,1] + -1.330;
   1:  PR[GP1:91,2] = PR[GP1:90,2] + -0.765;
   1:L PR[91] R[100]mm/sec CNT100;
   1:  PR[GP1:91,1] = PR[GP1:90,1] + -0.111;
   1:  PR[GP1:91,2] = PR[GP1:90,2] + -0.472;
   1:L PR[91] R[100]mm/sec CNT100;
   1:  PR[GP1:91,1] = PR[GP1:90,1] + 0.367;
   1:L PR[91] R[100]mm/sec CNT100;
   1:  PR[GP1:91,1] = PR[GP1:90,1] + 1.027;
   1:  PR[GP1:91,2] = PR[GP1:90,2] + -0.735;
   1:L PR[91] R[100]mm/sec CNT100;
   1:  PR[GP1:91,1] = PR[GP1:90,1] + 1.207;
   1:  PR[GP1:91,2] = PR[GP1:90,2] + -0.743;
   1:L PR[91] R[100]mm/sec CNT100;
   1:  PR[GP1:91,1] = PR[GP1:90,1] + 3.885;
   1:  PR[GP1:91,2] = PR[GP1:90,2] + -1.803;
   1:L PR[91] R[100]mm/sec CNT100;
   1:  PR[GP1:91,1] = PR[GP1:90,1] + 4.394;
   1:  PR[GP1:91,2] = PR[GP1:90,2] + -2.722;
   1:L PR[91] R[100]mm/sec CNT100;
   1:  PR[GP1:91,1] = PR[GP1:90,1] + 4.447;
   1:  PR[GP1:91,2] = PR[GP1:90,2] + -2.770;
   1:L PR[91] R[100]mm/sec CNT100;
   1:  PR[GP1:91,1] = PR[GP1:90,1] + 5.078;
   1:  PR[GP1:91,2] = PR[GP1:90,2] + -3.796;
   1:L PR[91] R[100]mm/sec CNT100;
   1:  PR[GP1:91,1] = PR[GP1:90,1] + 5.807;
   1:  PR[GP1:91,2] = PR[GP1:90,2] + -5.143;
   1:L PR[91] R[100]mm/sec CNT100;
   1:  PR[GP1:91,1] = PR[GP1:90,1] + 5.867;
   1:  PR[GP1:91,2] = PR[GP1:90,2] + -5.699;
   1:L PR[91] R[100]mm/sec CNT100;
   1:  PR[GP1:91,1] = PR[GP1:90,1] + 5.845;
   1:  PR[GP1:91,2] = PR[GP1:90,2] + -5.711;
   1:L PR[91] R[100]mm/sec CNT100;
   1:  PR[GP1:91,1] = PR[GP1:90,1] + 6.223;
   1:  PR[GP1:91,2] = PR[GP1:90,2] + -7.226;
   1:L PR[91] R[100]mm/sec CNT100;
   1:  PR[GP1:91,1] = PR[GP1:90,1] + 8.670;
   1:  PR[GP1:91,2] = PR[GP1:90,2] + -14.610;
   1:L PR[91] R[100]mm/sec CNT100;
   1:  PR[GP1:91,1] = PR[GP1:90,1] + 9.566;
   1:  PR[GP1:91,2] = PR[GP1:90,2] + -16.558;
   1:L PR[91] R[100]mm/sec CNT100;
   1:  PR[GP1:91,1] = PR[GP1:90,1] + 10.821;
   1:  PR[GP1:91,2] = PR[GP1:90,2] + -18.324;
   1:L PR[91] R[100]mm/sec CNT100;
   1:  PR[GP1:91,1] = PR[GP1:90,1] + 15.336;
   1:  PR[GP1:91,2] = PR[GP1:90,2] + -24.237;
   1:L PR[91] R[100]mm/sec CNT100;
   1:  PR[GP1:91,1] = PR[GP1:90,1] + 17.062;
   1:  PR[GP1:91,2] = PR[GP1:90,2] + -25.897;
   1:L PR[91] R[100]mm/sec CNT100;
   1:  PR[GP1:91,1] = PR[GP1:90,1] + 19.107;
   1:  PR[GP1:91,2] = PR[GP1:90,2] + -27.234;
   1:L PR[91] R[100]mm/sec CNT100;
   1:  PR[GP1:91,1] = PR[GP1:90,1] + 24.950;
   1:  PR[GP1:91,2] = PR[GP1:90,2] + -31.110;
   1:L PR[91] R[100]mm/sec CNT100;
   1:  PR[GP1:91,1] = PR[GP1:90,1] + 27.442;
   1:  PR[GP1:91,2] = PR[GP1:90,2] + -32.140;
   1:L PR[91] R[100]mm/sec CNT100;
   1:  PR[GP1:91,1] = PR[GP1:90,1] + 30.152;
   1:  PR[GP1:91,2] = PR[GP1:90,2] + -32.704;
   1:L PR[91] R[100]mm/sec CNT100;
   1:  PR[GP1:91,1] = PR[GP1:90,1] + 36.472;
   1:  PR[GP1:91,2] = PR[GP1:90,2] + -34.341;
   1:L PR[91] R[100]mm/sec CNT100;
   1:  PR[GP1:91,1] = PR[GP1:90,1] + 39.491;
   1:  PR[GP1:91,2] = PR[GP1:90,2] + -34.396;
   1:L PR[91] R[100]mm/sec CNT100;
   1:  PR[GP1:91,1] = PR[GP1:90,1] + 45.251;
   1:  PR[GP1:91,2] = PR[GP1:90,2] + -33.963;
   1:L PR[91] R[100]mm/sec CNT100;
   1:  PR[GP1:91,1] = PR[GP1:90,1] + 48.506;
   1:  PR[GP1:91,2] = PR[GP1:90,2] + -33.408;
   1:L PR[91] R[100]mm/sec CNT100;
   1:  PR[GP1:91,1] = PR[GP1:90,1] + 51.613;
   1:  PR[GP1:91,2] = PR[GP1:90,2] + -32.254;
   1:L PR[91] R[100]mm/sec CNT100;
   1:  PR[GP1:91,1] = PR[GP1:90,1] + 56.568;
   1:  PR[GP1:91,2] = PR[GP1:90,2] + -30.120;
   1:L PR[91] R[100]mm/sec CNT100;
   1:  PR[GP1:91,1] = PR[GP1:90,1] + 59.566;
   1:  PR[GP1:91,2] = PR[GP1:90,2] + -28.312;
   1:L PR[91] R[100]mm/sec CNT100;
   1:  PR[GP1:91,1] = PR[GP1:90,1] + 62.204;
   1:  PR[GP1:91,2] = PR[GP1:90,2] + -25.953;
   1:L PR[91] R[100]mm/sec CNT100;
   1:  PR[GP1:91,1] = PR[GP1:90,1] + 65.964;
   1:  PR[GP1:91,2] = PR[GP1:90,2] + -22.526;
   1:L PR[91] R[100]mm/sec CNT100;
   1:  PR[GP1:91,1] = PR[GP1:90,1] + 68.179;
   1:  PR[GP1:91,2] = PR[GP1:90,2] + -19.638;
   1:L PR[91] R[100]mm/sec CNT100;
   1:  PR[GP1:91,1] = PR[GP1:90,1] + 69.846;
   1:  PR[GP1:91,2] = PR[GP1:90,2] + -16.334;
   1:L PR[91] R[100]mm/sec CNT100;
   1:  PR[GP1:91,1] = PR[GP1:90,1] + 72.174;
   1:  PR[GP1:91,2] = PR[GP1:90,2] + -12.065;
   1:L PR[91] R[100]mm/sec CNT100;
   1:  PR[GP1:91,1] = PR[GP1:90,1] + 73.202;
   1:  PR[GP1:91,2] = PR[GP1:90,2] + -8.495;
   1:L PR[91] R[100]mm/sec CNT100;
   1:  PR[GP1:91,1] = PR[GP1:90,1] + 73.557;
   1:  PR[GP1:91,2] = PR[GP1:90,2] + -4.709;
   1:L PR[91] R[100]mm/sec CNT100;
   1:  PR[GP1:91,1] = PR[GP1:90,1] + 74.334;
   1:  PR[GP1:91,2] = PR[GP1:90,2] + -0.050;
   1:L PR[91] R[100]mm/sec CNT100;
   1:  PR[GP1:91,1] = PR[GP1:90,1] + 73.976;
   1:  PR[GP1:91,2] = PR[GP1:90,2] + 3.767;
   1:L PR[91] R[100]mm/sec CNT100;
   1:  PR[GP1:91,1] = PR[GP1:90,1] + 73.208;
   1:  PR[GP1:91,2] = PR[GP1:90,2] + 8.330;
   1:L PR[91] R[100]mm/sec CNT100;
   1:  PR[GP1:91,1] = PR[GP1:90,1] + 72.171;
   1:  PR[GP1:91,2] = PR[GP1:90,2] + 11.930;
